//Kommunikáció nyitás
IF NOT(GVL.bLaserCommOpen) THEN
	LaserSocketOpen(
		sSrvNetId:= '', 
		sRemoteHost:= sLaserRemoteHost, 
		nRemotePort:= 20001, 
		bExecute:= bLaserSocketOpenEnable, 
		tTimeout:= T#45S, 
		bBusy=> bLaserSocketbusy, 
		bError=> bLaserSocketError, 
		nErrId=> nLaserSocketErrId, 
		hSocket=> hLaserSocket);
	IF bLaserSocketOpenEnable THEN
		IF (NOT(bLaserSocketError) AND NOT(bLaserSocketError) AND NOT(bLaserSocketbusy)) THEN
			bLaserSocketOpenEnable := FALSE;
			GVL.bLaserCommOpen:=TRUE;
			LaserSocketOpen(
				sSrvNetId:= '', 
				sRemoteHost:= sLaserRemoteHost, 
				nRemotePort:= 5000, 
				bExecute:= FALSE, 
				tTimeout:= T#45S, 
				bBusy=> bLaserSocketbusy, 
				bError=> bLaserSocketError, 
				nErrId=> nLaserSocketErrId, 
				hSocket=> hLaserSocket);
		ELSE
			IF NOT(bLaserSocketbusy) THEN
				bLaserSocketOpenEnable:=FALSE;
			END_IF
		END_IF
	ELSE
		bLaserSocketOpenEnable:=TRUE;
	END_IF
END_IF

// Parancsfordítások a lézer számára
IF bLaserSendReady=TRUE THEN				// a parancsküldés befejeződött,
	IF s_InCommand='GETJOB' THEN
		sLaserSend:='GetJob;';
	END_IF
	IF s_InCommand='START' THEN
		sLaserSend:='Start;';
	END_IF
	IF s_InCommand='SETTYPE' THEN
		s_TypeCode:=TO_STRING(GVL.iSelectedProductType);
		sLaserSend:=CONCAT('SetVars;TypeCode;',CONCAT(s_TypeCode,';'));
	END_IF
	IF s_InCommand='GETSTATUS' THEN
		sLaserSend:='GetStatus;';
	END_IF
	IF s_InCommand='RECEIVE' THEN
		bLaserSocketReceiveRequest:=TRUE;
		bLaserSendReady:=FALSE;
		sLaserReceived:='';
	END_IF
END_IF

// Csak akkor próbáljon kommunikálni, ha már megnyílt a kapcsolat
IF GVL.bLaserCommOpen=TRUE THEN
	// Adatküldés, ha van mit küldeni
	IF sLaserSend<>'' THEN
		IF bLaserSocketSendEnable THEN
			bLaserSocketSendEnable:=FALSE;
			sLaserSend:='';
			bLaserSocketReceiveRequest:=TRUE; // Választ is várunk majd a lézertől.
		ELSE
			MEMSET(ADR(baReceivedByteArray), 0, 256);
			MEMSET(ADR(baSendByteArray), 0, 256);
			baSendByteArray := MAXSTRING_TO_BYTEARR(sLaserSend);
			uSendByteLen := INT_TO_UDINT(LEN(sLaserSend));
			baSendByteArray[uSendByteLen]:=16#D;
			baSendByteArray[uSendByteLen+1]:=16#A;
			bLaserSocketSendEnable:=TRUE;
			bLaserSendReady:=FALSE;
			sLaserReceived:='';
		END_IF;
		LaserSocketSend(
			sSrvNetId:= '', 
			hSocket:= hLaserSocket, 
			cbLen:= uSendByteLen + 2, 
			pSrc:= ADR(baSendByteArray), 
			bExecute:= bLaserSocketSendEnable, 
			tTimeout:= T#5S, 
			bBusy=> bLaserSocketbusy, 
			bError=> bLaserSocketError, 
			nErrId=> nLaserSocketErrId);
	END_IF
	// Ha van adatfogadási igény, akkor minden páros ciklusnál indítson adatfogadást
	IF (bLaserSocketReceiveRequest=TRUE) AND (bEvenCycle=TRUE) THEN
		bLaserSocketReceiveEnable:=TRUE;
	ELSE
		bLaserSocketReceiveEnable:=FALSE;		
	END_IF
	//Adatfogadás, ha van rá parancs
	LaserSocketReceive(
		sSrvNetId:= '', 
		hSocket:= hLaserSocket, 
		cbLen:= 255, 
		pDest:= ADR(baReceivedByteArray), 
		bExecute:= bLaserSocketReceiveEnable, 
		tTimeout:= T#5S, 
		bBusy=> bLaserSocketbusy, 
		bError=> bLaserSocketError, 
		nErrId=> nLaserSocketErrId, 
		nRecBytes=> nLaserReceivedBytesNum);
	IF baReceivedByteArray[0]>0 THEN // Ha érkezett válasz a lézertől, akkor
		nLaserReceivedBytesNum:=0;	// töröljük, hogy ne lépjen be ide újra,
		bLaserSocketReceiveRequest:=FALSE;	// ne várjon több válaszra,		
		bLaserSendReady:=TRUE;				// a parancsküldés befejeződött, töröljük a parancsot, és
		bLaserSendOK:=(baReceivedByteArray[0]=16#6); // ha ACK jel jött, akkor OK.
		sLaserReceived := BYTEARR_TO_MAXSTRING(baReceivedByteArray);
		IF sLaserReceived='$06;0000;$R$N' THEN
			s_InCommand:='';
		ELSE
			s_InCommand:=CONCAT('LÉZER HIBA: ',sLaserReceived);
		END_IF
	END_IF

	//Kommunikáció bontás
	LaserSocketClose(
		sSrvNetId:= '', 
		hSocket:= hLaserSocket, 
		bExecute:= bLaserSocketCloseEnable, 
		tTimeout:= T#45S, 
		bBusy=> bLaserSocketbusy, 
		bError=> bLaserSocketError, 
		nErrId=> nLaserSocketErrId);

	bEvenCycle:=NOT bEvenCycle;
END_IF

END_PROGRAM

// ---- POUs/PISTI/Components/TEST_R_INTERPOL.TcPOU
PROGRAM TEST_R_INTERPOL
VAR
	rRNTC_MIN0, rRNTC_MIN1, rRNTC_MAX0, rRNTC_MAX1, rPt_MIN, rPt_MAX, rT: REAL;
END_VAR

rRNTC_MIN0:=f_GetNTCMinR(rTemp:=rT, nProd:=0);
rRNTC_MAX0:=f_GetNTCMaxR(rTemp:=rT, nProd:=0);
rRNTC_MIN1:=f_GetNTCMinR(rTemp:=rT, nProd:=1);
rRNTC_MAX1:=f_GetNTCMaxR(rTemp:=rT, nProd:=1);
rPt_MIN:=f_GetPtMinR(rTemp:=rT);
rPt_MAX:=f_GetPtMaxR(rTemp:=rT);

END_PROGRAM

// ---- POUs/PISTI/Helpers/f_GetNTCNomR.TcPOU
FUNCTION f_GetNTCNomR : real
VAR_INPUT
	rTemp: REAL;
	nProd: UINT;
END_VAR
VAR
	nI: INT;
	rT0, rT1, rR0, rR1, rM: REAL;
END_VAR
VAR CONSTANT
	rCorr: REAL := 1.1;
	NTC_Sensing_MinRT: ARRAY[0..1, 0..25] OF REAL := 
	[15, 16, 17, 18, 19, 20, 21, 22, 23, 24, 25, 26, 27, 28, 29, 30, 31, 32, 33, 34, 35, 36, 37, 38, 39, 40,
	14966.9, 14299.6, 13665.8, 13063.7, 12491.4, 11947.3, 11430, 10937.9, 10469.8, 10024.2, 9600, 9188.1, 8796.1, 8423, 8067.6, 7729.2, 7406.8, 7099.6, 6806.7, 6527.5, 6261.3, 6007.2, 5764.9, 5533.6, 5312.7, 5101.9];
	NTC_GE_MinRT: ARRAY[0..1, 0..23] OF REAL := 
	[15, 16, 17, 18, 19, 20, 21, 22, 23, 24, 25, 26, 27, 28, 29, 30, 31, 32, 33, 34, 35, 36, 38, 40,
	15133, 14457, 13815, 13206, 12626, 12075, 11552, 11053, 10579, 10128, 9700, 9279.9, 8883.4, 8506.1, 8146.8, 7804.7, 7478.7, 7168.1, 6872.1, 6589.9, 6320.7, 6064, 5585.4, 5149.3];
END_VAR

nI:=1;
(*IF nProd=0 THEN
	WHILE (NTC_Sensing_MinRT[0,nI]<rTemp) AND (nI<25) DO
		nI:=nI+1;
	END_WHILE
	rT0:=NTC_Sensing_MinRT[0,nI-1];
	rT1:=NTC_Sensing_MinRT[0,nI];
	rR0:=NTC_Sensing_MinRT[1,nI-1];
	rR1:=NTC_Sensing_MinRT[1,nI];
	rM:=(rR1-rR0)/(rT1-rT0);
	f_GetNTCMinR:=rR0+rM*(rTemp-rT0);
ELSE
	WHILE (NTC_GE_MinRT[0,nI]<rTemp) AND (nI<23) DO
		nI:=nI+1;
	END_WHILE
	rT0:=NTC_GE_MinRT[0,nI-1];
	rT1:=NTC_GE_MinRT[0,nI];
	rR0:=NTC_GE_MinRT[1,nI-1];
	rR1:=NTC_GE_MinRT[1,nI];
	rM:=(rR1-rR0)/(rT1-rT0);
	f_GetNTCMinR:=rR0+rM*(rTemp-rT0);	
END_IF*)
WHILE (GVL.NTC_Sensing_NomRT[0,nI]<rTemp) AND (nI<25) DO
	nI:=nI+1;
END_WHILE
rT0:=GVL.NTC_Sensing_NomRT[0,nI-1];
rT1:=GVL.NTC_Sensing_NomRT[0,nI];
rR0:=GVL.NTC_Sensing_NomRT[1,nI-1];
rR1:=GVL.NTC_Sensing_NomRT[1,nI];
rM:=(rR1-rR0)/(rT1-rT0);
f_GetNTCMinR:=(rR0+rM*(rTemp-rT0))/(1+GVL.rNTCDev/100);

END_FUNCTION

// ---- POUs/PISTI/Helpers/f_GetPtNomR.TcPOU
FUNCTION f_GetPtNomR : real
VAR_INPUT
	rTemp: REAL := 25;
END_VAR
VAR
	nI: INT;
	rT0, rT1, rR0, rR1, rM: REAL;
END_VAR
VAR CONSTANT
	Pt_MinRT: ARRAY[0..1, 0..15] OF REAL := 
	[0,20,40,60,80,100,120,140,160,180,200,220,240,260,280,300,
	990,1067,1143,1219,1294,1368,1442,1516,1588,1661,1733,1804,1875,1945,2015,2084];
END_VAR

nI:=1;
WHILE (Pt_MinRT[0,nI]<rTemp) AND (nI<15) DO
	nI:=nI+1;
END_WHILE
rT0:=Pt_MinRT[0,nI-1];
rT1:=Pt_MinRT[0,nI];
rR0:=Pt_MinRT[1,nI-1];
rR1:=Pt_MinRT[1,nI];
rM:=(rR1-rR0)/(rT1-rT0);
f_GetPtMinR:=rR0+rM*(rTemp-rT0);

END_FUNCTION

// ---- POUs/PISTI/Helpers/f_GetPtTfromR.TcPOU
FUNCTION f_GetPtTfromR : real
VAR_INPUT
	rR: REAL;
END_VAR
VAR
	nI: INT;
	rT0, rT1, rR0, rR1, rM: REAL;
END_VAR
VAR CONSTANT
	Pt_RT: ARRAY[0..1, 0..15] OF REAL := 
	[0,20,40,60,80,100,120,140,160,180,200,220,240,260,280,300,
	1000,1077.9,1155.4,1232.4,1309,1385.1,1460.7,1535.8,1610.5,1684.8,1758.6,1831.9,1904.7,1977.1,2049.1,2120.5];
END_VAR

nI:=1;
WHILE (Pt_RT[1,nI]<rR) AND (nI<15) DO
	nI:=nI+1;
END_WHILE
rT0:=Pt_RT[0,nI-1];
rT1:=Pt_RT[0,nI];
rR0:=Pt_RT[1,nI-1];
rR1:=Pt_RT[1,nI];
rM:=(rT1-rT0)/(rR1-rR0);
f_GetPtTfromR:=rT0+rM*(rR-rR0);

END_FUNCTION

// ---- POUs/PISTI/Helpers/f_GetISOLvalue.TcPOU
FUNCTION f_GetISOLvalue : REAL
VAR_INPUT
	rVoltage : REAL;
END_VAR
VAR
	rVoltagePerOhmRate : REAL := 5100/0.889;
END_VAR

f_GetISOLvalue := rVoltage * rVoltagePerOhmRate;

END_FUNCTION

// ---- GlobalTextList.TcGTLO
TEXTLIST GlobalTextList
  140 = ''
  845 = '\nFizikális gombok használata NTC vágáshoz.\nZöld gomb: NTC vágófej le-fel\nPiros gomb: NTC vágófej le-fel'
  844 = '\nFizikális gombok használata NTC vágáshoz.Zöld gomb: NTC vágófej le-fel\nPiros gomb: NTC vágófej le-fel'
  841 = '\nZöld gomb: NTC vágófej le-fel\nPiros gomb: NTC vágófej le-fel'
  842 = '\nZöld gomb: NTC vágás\nPiros gomb: NTC elengedés'
  840 = '\nZöld gomb: NTC vágófej le-fel\nPiros gomb: NTC vágófej le-fel'
  43 = '%'
  47 = '%./100'
  45 = '%.1f'
  46 = '%.2f'
  48 = '%/100'
  157 = '%c'
  130 = '%d'
  60 = '%f'
  59 = '%lr'
  58 = '%s'
  73 = '%u'
  368 = "'ELEKTRÓDA$R$NCSERE!'"
  49 = '.1f'
  2499 = '1. elektróda pár'
  807 = '1. elektródapár'
  717 = '1. heg.'
  380 = '1. HEGESZTESHEZ'
  390 = '1. hegesztés program'
  384 = '1. HEGESZTÉSHEZ'
  800 = '1. VÉGPOZÍCIÓ'
  802 = '1. VÉGPOZÍCIÓHOZ'
  41 = '11'
  44 = '1f'
  7390 = '2. elektróda pár'
  809 = '2. elektródapár'
  718 = '2. heg.'
  381 = '2. HEGESZTESHEZ'
  391 = '2. hegesztés program'
  385 = '2. HEGESZTÉSHEZ'
  801 = '2. VÉGPOZÍCIÓHOZ'
  5960 = '3. elektróda pár'
  808 = '3. elektródapár'
  719 = '3. heg.'
  382 = '3. HEGESZTESHEZ'
  392 = '3. hegesztés program'
  386 = '3. HEGESZTÉSHEZ'
  317 = '4. heg.'
  287 = '4. heg. deformációja:'
  383 = '4. HEGESZTESHEZ'
  708 = '4. hegesztés'
  286 = '4. hegesztés deformációja:'
  393 = '4. hegesztés program'
  710 = '4. hegesztés, STOP érték [um]:'
  387 = '4. HEGESZTÉSHEZ'
  318 = '5. heg.'
  288 = '5. heg. deformációja:'
  709 = '5. hegesztés'
  394 = '5. hegesztés program'
  711 = '5. hegesztés, STOP érték [um]:'
  388 = '5. HEGESZTÉSHEZ'
  484 = '6 s'
  729 = '6. hegesztés program'
  341 = '6.0'
  116 = '600V'
  115 = '600VBe'
  117 = '600VExt'
  314 = '637 GYÁRTÓ CELLA'
  6089 = '637900'
  730 = '7. hegesztés program'
  9321 = '745900'
  7231 = '745910'
  830 = '<!> db'
  509 = 'A jelölö lézer saját vezérlö szoftvere'
  504 = 'A jelölő lézer saját vezérlő szoftvere'
  901 = 'A Pt oldali kamera saját vezérlő szoftvere'
  637 = 'A tengelypozíciók a megfelelö\nszervízfüleken állíthatók be.\n\nAz alábbi gombok a megfelelö \nszervízfülre navigálnak:'
  625 = 'A tengelypozíciók a megfelelő\nszervízfüleken állíthatók be.\n\nAz alábbi gombok a megfelelő \nszervízfülre navigálnak:'
  619 = 'A tengelypozíciók a megfelelő\nszervízfüleken állíthatók be.\nAz alábbi gombok a\nmegfelelő szervízfülre\nnavigálnak:'
  620 = 'A tengelypozíciók a megfelelő\nszervízfüleken állíthatók be.\nAz alábbi gombok a \nmegfelelő szervízfülre\nnavigálnak:'
  622 = 'A tengelypozíciók a megfelelő\nszervízfüleken állíthatók be.\nAz alábbi gombok a megfelelő\nszervízfülre\nnavigálnak:'
  623 = 'A tengelypozíciók a megfelelő\nszervízfüleken állíthatók be.\nAz alábbi gombok a megfelelő \nszervízfülre\nnavigálnak:'
  624 = 'A tengelypozíciók a megfelelő\nszervízfüleken állíthatók be.\nAz alábbi gombok a megfelelő \nszervízfülre navigálnak:'
  621 = 'A tengelypozíciók a megfelelő\nszervízfüleken állíthatók be.\nAz alábbi gombok a megfelelő szervízfülre\nnavigálnak:'
  618 = 'A tengelypozíciók a megfelelő szervízfüleken állíthatók be. Az alábbi gombok a megfelelő szervízfülre navigálnak:'
  62 = 'Act. Pos:'
  8 = 'AdapterLefogó'
  544 = 'Adapterlefogó'
  5 = 'AdapterLefogóBent'
  4 = 'AdapterLefogóKint'
  818 = 'Adapterérzékelö'
  2 = 'Adapterérzékelő'
  917 = 'ADD/DELETE USER'
  300 = 'Admin'
  79 = 'AEH'
  1962 = 'AJTÓ\nZÁR'
  692 = 'Ajtók zárva'
  143 = 'ALARM'
  352 = 'Alsó rész'
  179 = 'AUTO'
  285 = 'AUTO STOP'
  488 = 'Automata'
  713 = 'Automatikus mentés'
  81 = 'AVH'
  771 = 'bal fent'
  832 = 'Bal fék'
  772 = 'bal lent'
  838 = 'Bal lábérzékelö'
  833 = 'Bal lábérzékelő'
  425 = 'Bal pofa'
  105 = 'Balon'
  436 = 'Balra'
  439 = 'Be'
  20 = 'Behelyezés'
  547 = 'BEHELYEZÉS'
  668 = 'Belépve, mint:'
  669 = 'BELÉPVE, MINT:'
  107 = 'Bent'
  591 = 'Beragadt TCP IP kapcsolatok törölve'
  97 = 'Bereit'
  465 = 'BEZÁR'
  826 = 'BEÁLLÍTÁS'
  348 = 'Beállítások'
  714 = 'Beállítások automatikus mentése'
  682 = 'BIZTONSÁGI AJTÓ RETESZ'
  679 = 'Biztonsági kör OK'
  678 = 'Biztonsági relé föld OK'
  677 = 'Biztonsági relé táp OK'
  676 = 'Biztonsági rendszer'
  4978 = 'Biztos?'
  876 = 'Busy'
  900 = 'Checker indítása'
  794 = 'Ciklusok'
  160 = 'CLOSE'
  122 = 'Com Open'
  878 = 'Comm Open'
  266 = 'COMMUNICATION OPEN'
  865 = 'Csatlakozó'
  4888 = 'Csatlakozó\nfedél csukva'
  491 = 'Csatlakozó\nfedél nyitva'
  6459 = 'Csatlakozó\nfedél zárva'
  866 = 'Csatlakozó (745)'
  864 = 'Csatlakozó fedél'
  490 = 'Csatlakozó fedél edelNyitva?'
  532 = 'CSIPESZ NYIT'
  531 = 'CSIPESZ ZÁR'
  277 = 'DARABSZÁM'
  812 = 'db'
  707 = 'Deformációalapú hegesztés-leállítás'
  4104 = 'Dolgozói szám'
  814 = 'Elekróda karbantartás'
  805 = 'ELEKT-\nRÓDA-\nTISZTÍTÁS'
  208 = 'Elektroden\nAnfordem'
  96 = 'ElektrodenAnfordem'
  364 = 'ELEKTRÓDA  CSERE!'
  363 = 'ELEKTRÓDA CSERE!'
  365 = 'ELEKTRÓDA RÉGI'
  366 = 'ELEKTRÓDA$R$NCSERE!'
  370 = 'ELEKTRÓDACSERE'
  369 = 'ELEKTRÓDACSERE!'
  803 = 'ELEKTRÓDATISZT'
  804 = 'ELEKTRÓDATISZTÍTÁS'
  367 = 'ELEKTRÓDA\\R\\NCSERE!'
  907 = 'ELFOGADHATÓ'
  222 = 'ELLENALLAS'
  252 = 'ELLENALLAS ETALON'
  450 = 'ELLENÁLLÁS'
  452 = 'Ellenállás'
  451 = 'ELLENÁLLÁS ETALON'
  658 = 'Eltelt idö'
  480 = 'Eltelt idö (s)'
  513 = 'Elvárt kód:'
  469 = 'ELVÁRT:'
  379 = 'Elvégzendö müveletek'
  347 = 'Elvégzendö műveletek'
  516 = 'ELÖHAJLÍTASHOZ'
  424 = 'ELÖHAJLÍTÁS'
  517 = 'ELÖHAJLÍTÁSHOZ'
  349 = 'Elöhajlító'
  83 = 'ELŐHAJLITASHOZ'
  194 = 'ELŐHAJLÍTÁS'
  76 = 'Előhajlító'
  77 = 'Előhajlító fent'
  546 = 'Enged'
  701 = 'EPSON RC+ megnyitása'
  410 = 'Eredmény:'
  466 = 'EREDMÉNYEK'
  174 = 'ERROR'
  246 = 'Error'
  877 = 'Error ID'
  283 = 'Error reset'
  175 = 'ESTOP'
  695 = 'Etalon'
  556 = 'Etalon mérés'
  694 = 'ETALON MÉRÉS'
  109 = 'FedelLecsukva?'
  249 = 'FedelNyitva?'
  829 = 'FEDÉL'
  78 = 'FEH'
  431 = 'Fej le'
  670 = 'FEJLESZTÖ'
  716 = 'Felfüggeszt'
  350 = 'Felsö rész'
  103 = 'Fent'
  779 = 'fent'
  775 = 'fent bent'
  776 = 'fent kint'
  725 = 'Fizikális gombok használata NTC vágáshoz.\nZöld gomb: NTC vágás\nPiros gomb: NTC elengedés'
  846 = 'Fizikális gombok használata NTC vágáshoz.\nZöld gomb: NTC vágófej le-fel\nPiros gomb: NTC vágófej le-fel'
  503 = 'FOBA Draw indítása'
  268 = 'Fogadott:'
  269 = 'Fogadás'
  42 = 'fok'
  690 = 'FOLYTAT'
  554 = 'Forgásirány:'
  149 = 'Forward'
  909 = 'FRISSÍT'
  80 = 'FVH'
  3 = 'Fénykapu'
  674 = 'FÉNYSOROMPÓ'
  434 = 'Fütötömb'
  527 = 'Fütötömb\nfelfütött'
  478 = 'Fütötömb beállított\nhömérséklete (C)'
  615 = 'Fütötömb beállított\nhömérséklete (C):'
  656 = 'Fütötömb beállított\nhömérséklete [C]'
  644 = 'Fütötömb beállított \nhömérséklete (C):'
  650 = 'Fütötömb beállított \nhömérséklete [C]:'
  477 = 'Fütötömb hömérséklete (C)'
  67 = 'Főnök'
  530 = 'GroupBox'
  291 = 'Hajlítás'
  354 = 'Hajlítók'
  316 = 'Heg. deformációja:'
  904 = 'Hegesz-\ntéshez'
  795 = 'HEGESZ-\nTÖFEJ\nTISZTÍTÁS'
  903 = 'Hegesz-téshez'
  85 = 'HEGESZTES1HEZ'
  87 = 'HEGESZTES2HOZ'
  86 = 'HEGESZTES2HÖZ'
  88 = 'HEGESZTES3HOZ'
  89 = 'HEGESZTES4HEZ'
  90 = 'HEGESZTES5HÖZ'
  138 = 'HEGESZTESHEZ'
  216 = 'HEGESZTESHEZ1'
  217 = 'HEGESZTESHEZ2'
  21 = 'Hegesztés'
  74 = 'HEGESZTÉS'
  791 = 'HEGESZTÉS KÉSZ'
  292 = 'Hegesztés1'
  627 = 'HEGESZTÉS1'
  519 = 'HEGESZTÉS1-HEZ'
  293 = 'Hegesztés2'
  628 = 'HEGESZTÉS2'
  520 = 'HEGESZTÉS2-HÖZ'
  294 = 'Hegesztés3'
  629 = 'HEGESZTÉS3'
  521 = 'HEGESZTÉS3-HOZ'
  295 = 'Hegesztés4'
  630 = 'HEGESZTÉS4'
  522 = 'HEGESZTÉS4-HEZ'
  296 = 'Hegesztés5'
  631 = 'HEGESZTÉS5'
  523 = 'HEGESZTÉS5-HÖZ'
  305 = 'Hegesztés6'
  306 = 'Hegesztés7'
  902 = 'Hegesztéshez'
  588 = 'Hegesztö'
  799 = 'Hegesztö elektróda karbantartás'
  407 = 'Hegesztö státusz'
  579 = 'Hegesztö üzemkész'
  459 = 'HEGESZTÖFEJ\nTISZTÍTÁS'
  781 = 'Hegesztöfej I/O-k'
  400 = 'HEGESZTÖFEJ TISZT.'
  783 = 'Hegesztöfej1'
  757 = 'Hegesztöfej1 bal fent'
  761 = 'Hegesztöfej1 bal lent'
  758 = 'Hegesztöfej1 jobb fent'
  762 = 'Hegesztöfej1 jobb lent'
  755 = 'Hegesztöfej1 le'
  765 = 'Hegesztöfej1 útmérö:'
  784 = 'Hegesztöfej2'
  756 = 'Hegesztöfej2 be'
  763 = 'Hegesztöfej2 fent bent'
  759 = 'Hegesztöfej2 fent kint'
  770 = 'Hegesztöfej2 ki'
  764 = 'Hegesztöfej2 lent bent'
  760 = 'Hegesztöfej2 lent kint'
  766 = 'Hegesztöfej2 útmérö:'
  785 = 'Hegesztöfej3'
  768 = 'Hegesztöfej3 fent'
  767 = 'Hegesztöfej3 le'
  769 = 'Hegesztöfej3 lent'
  593 = 'Hegesztöfejek alapállapotban'
  356 = 'Hegesztögép státusza'
  9 = 'Hegesztő'
  68 = 'Hegesztő1'
  71 = 'Hegesztő1 Útmérő:'
  735 = 'Hegesztő1 útmérő:'
  69 = 'Hegesztő2'
  72 = 'Hegesztő2 Útmérő:'
  736 = 'Hegesztő2 útmérő:'
  70 = 'Hegesztő3'
  274 = 'HEGESZTŐFEJ TISZT.'
  739 = 'Hegesztőfej1 bal fent'
  740 = 'Hegesztőfej1 bal lent'
  743 = 'Hegesztőfej1 fent kint'
  741 = 'Hegesztőfej1 jobb fent'
  742 = 'Hegesztőfej1 jobb lent'
  750 = 'Hegesztőfej1 le'
  737 = 'Hegesztőfej1 útmérő:'
  751 = 'Hegesztőfej2 be'
  745 = 'Hegesztőfej2 fent bent'
  744 = 'Hegesztőfej2 fent kint'
  747 = 'Hegesztőfej2 lent bent'
  746 = 'Hegesztőfej2 lent kint'
  738 = 'Hegesztőfej2 útmérő:'
  753 = 'Hegesztőfej3 bal fent'
  754 = 'Hegesztőfej3 bal lent'
  748 = 'Hegesztőfej3 fent'
  752 = 'Hegesztőfej3 le'
  749 = 'Hegesztőfej3 lent'
  6 = 'HegesztőFent'
  7 = 'HegesztőLent'
  782 = 'Hello'
  732 = 'HIBA'
  398 = 'Hiba kód:'
  399 = 'Hiba törlés'
  403 = 'Hiba törlése'
  401 = 'Hibakód:'
  404 = 'Hibatörlés'
  733 = 'HIBATÖRLÉS'
  279 = 'HIBÁS'
  857 = 'Himba'
  867 = 'Himba alapállapotban'
  858 = 'Himba be'
  860 = 'Himba elöl'
  861 = 'Himba hátul'
  870 = 'Himba OK'
  863 = 'Himba pozíció'
  859 = 'Himba érzékelő'
  862 = 'HIMBÁHOZ'
  53 = 'HOME'
  449 = 'HÖM (C)'
  332 = 'HÖM [C]'
  529 = 'Hömérséklet (C)'
  910 = 'Hüvely poz OK'
  911 = 'Hüvely pozíció'
  912 = 'Hüvely van'
  721 = 'Hüvelyek OK'
  448 = 'HŐM (C)'
  321 = 'HŐM MEAS (C)'
  214 = 'Hőmérséklet'
  218 = 'Hőmérséklet (C)'
  224 = 'IDOALLANDO'
  250 = 'IDOALLANDO_OK'
  323 = 'IDÖÁLLANDÓ'
  485 = 'Idöállandó'
  642 = 'Idöállandó\nfelsö határa:'
  616 = 'Idöállandó\nfelső határa:'
  647 = 'Idöállandó \nfelsö határa (s):'
  648 = 'Idöállandó \nfelsö határa [s]:'
  645 = 'Idöállandó \nfelsö határa:'
  481 = 'Idöállandó (s)'
  328 = 'IDÖÁLLANDÓ [s]'
  654 = 'Idöállandó [s]'
  298 = 'IDÖÁLLANDÓ_OK'
  242 = 'Időállandó (s)'
  4983 = 'IGEN'
  789 = 'In-Sight Explorer indítása'
  358 = 'INDÍTÁS'
  817 = 'Indítás fénysorompóval'
  787 = 'Indítási feltételek'
  585 = 'Indítási opciók'
  170 = 'INIT'
  324 = 'ISOL'
  221 = 'ISOL_OK'
  672 = 'IV-Navigator indítása'
  223 = 'IZOLÁCIÓ'
  114 = 'Izolációs érték'
  243 = 'Izolációs érték (V)'
  232 = 'Izolációs érték(V)'
  311 = 'JELENLEGI FOLYAMAT:'
  389 = 'Jelenlegi pozíció:'
  825 = 'Jelenlegi érték [%]:'
  824 = 'Jelenlegi érték [0...100 %]:'
  325 = 'JELÖLÉS'
  297 = 'JELÖLÉS_OK'
  773 = 'jobb fent'
  835 = 'Jobb fék'
  774 = 'jobb lent'
  839 = 'Jobb lábérzékelö'
  834 = 'Jobb lábérzékelő'
  426 = 'Jobb pofa'
  106 = 'Jobbon'
  55 = 'JOG +'
  56 = 'JOG -'
  4109 = 'Jogosultság'
  181 = 'JozsiProcess.asActualProgram[0,INDEX]'
  182 = 'JozsiProcess.asActualProgram[1,INDEX]'
  183 = 'JozsiProcess.asActualProgram[2,INDEX]'
  184 = 'JozsiProcess.asActualProgram[3,INDEX]'
  185 = 'JozsiProcess.asActualProgram[4,INDEX]'
  186 = 'JozsiProcess.asActualProgram[5,INDEX]'
  64 = 'JozsiTengely'
  278 = 'JÓ'
  24 = 'Józsi'
  604 = 'Kamera'
  728 = 'KAMERA'
  895 = 'Kamera Adapter'
  893 = 'Kamera All pass'
  894 = 'Kamera Any fail'
  886 = 'Kamera Aquiring'
  890 = 'Kamera Inspect toggle'
  889 = 'Kamera Inspecting'
  896 = 'Kamera Kappe'
  888 = 'Kamera Online'
  892 = 'Kamera Part Detected'
  727 = 'Kamera pozíció'
  897 = 'Kamera Pt'
  891 = 'Kamera Results available'
  898 = 'Kamera Run'
  882 = 'Kamera Set Offline'
  887 = 'Kamera Setup'
  881 = 'Kamera Trigger'
  885 = 'Kamera Trigger Ack'
  880 = 'Kamera Trigger EN'
  884 = 'Kamera Trigger Ready'
  723 = 'KAMERA-\nEREDMÉNYEK'
  610 = 'Kamera1'
  611 = 'Kamera2'
  722 = 'KAMERAEREDMÉNYEK'
  724 = 'Kameravizsgálat\neredménye'
  726 = 'KAMERÁHOZ'
  165 = 'KAPPE'
  251 = 'Kappe Pistikének'
  432 = 'Kappe prés'
  464 = 'KAPPE PRÉS'
  307 = 'Kappe, robot'
  15 = 'KappeBal'
  13 = 'KappeBalFent'
  14 = 'KappeBalLent'
  12 = 'KappeFelLe'
  10 = 'KappeFent'
  18 = 'KappeJobb'
  16 = 'KappeJobbFent'
  17 = 'KappeJobbLent'
  11 = 'KappeLent'
  337 = 'KappeNincsLent'
  137 = 'KAPPEZASHOZ'
  905 = 'Kappé-\nzáshoz'
  22 = 'Kappézás'
  634 = 'KAPPÉZÁS'
  525 = 'KAPPÉZÁSHOZ'
  798 = 'KARBANTARTÁS'
  855 = 'Keyence SR-1000W'
  856 = 'Keyence SR-1000W/ nem Zebra'
  693 = 'Ki'
  417 = 'Kieg. müveletek'
  416 = 'Kiegészítö müveletek'
  346 = 'KILÉPÉS'
  3792 = 'Kilépés'
  108 = 'Kint'
  152 = 'Kiszedo'
  376 = 'Kiszedö'
  351 = 'Kitol'
  299 = 'KIÉRTÉKELÉS'
  422 = 'Kommunikáció'
  557 = 'KOMMUNIKÁCIÓS CSATORNA MEGNYITVA'
  505 = 'KOMMUNIKÁCIÓS VONAL MEGNYITVA'
  608 = 'Kábeltáv OK'
  688 = 'Kérem, adja meg a vonalkód\nolvasó\nsegítségével a gyártani kívánt terméktípust!\nÜgyeljen rá, hogy a megfelelő NTC és Pt1000\nalkatrészek legyenek betárazva, felhasználva!\nHa kell, ezek vonalkódját is be lehet olvastatni.'
  687 = 'Kérem, adja meg a vonalkód\nolvasó segítségével\na \ngyártani kívánt terméktípust!\nÜgyeljen rá, hogy a megfelelő NTC és Pt1000\nalkatrészek legyenek betárazva, felhasználva!\nHa kell, ezek vonalkódját is be lehet olvastatni.'
  686 = 'Kérem, adja meg a vonalkód\nolvasó segítségével a \ngyártani kívánt terméktípust!\nÜgyeljen rá, hogy a megfelelő NTC és Pt1000 alkatrészek legyenek betárazva, felhasználva!\nEzek vonalkódját is be lehet olvastatni.'
  685 = 'Kérem, adja meg a vonalkód\nolvasó segítségével a \ngyártani kívánt terméktípust!\nÜgyeljen rá, hogy a megfelelő NTC és Pt1000 alkatrészek legyenek betárazva, felhasználva! Ezek vonalkódját is be lehet olvastatni.'
  684 = 'Kérem, adja meg a vonalkód\nolvasó segítségével a\ngyártani kívánt terméktípust!'
  689 = 'Kérem, adja meg a vonalkódolvasó\nsegítségével a gyártani kívánt terméktípust!\nÜgyeljen rá, hogy a megfelelő NTC és Pt1000\nalkatrészek legyenek betárazva, felhasználva!\nHa kell, ezek vonalkódját is be lehet olvastatni.'
  471 = 'Kérem, indítás elött ellenörízze,\nhogy idegen tárgyaktól\nmentes-e a munkatér, és\nminden készen áll-e az indításra!'
  470 = 'Kérem, indítás előtt ellenörízze,\nhogy idegen tárgyaktól\nmentes-e a munkatér, és\nminden készen áll-e az indításra!'
  699 = 'Kérem, tegye be a(z) %s. etalont,\nmajd nyomja meg a START gombot!'
  698 = 'Kérem, tegye be az %s. etalont,\nmajd nyomja meg a START gombot!'
  700 = 'Kérem, tegye be az ETALON%s-t,\nmajd nyomja meg a START gombot!'
  156 = 'Kérleltetés'
  372 = 'Késleltetés'
  359 = 'KÉSZ'
  395 = 'Készenléti program'
  444 = 'Kézi'
  823 = 'Kívánt érték [0...100 %]:'
  822 = 'Kívánt érték:'
  336 = 'Kódolvasó'
  514 = 'KÓDOLVASÓ'
  852 = 'KÓDOLVASÓ 2'
  333 = 'KÓDOLVASÓHOZ'
  853 = 'KÓDOLVASÓHOZ 2'
  256 = 'Következő lépés'
  272 = 'Közvetett parancs'
  273 = 'Közvetlen parancs'
  267 = 'Küld:'
  506 = 'kÜLDÉS'
  827 = 'KÜLDÉS'
  1 = 'Label'
  435 = 'Le'
  828 = 'LEKÉRDEZÉS'
  104 = 'Lent'
  780 = 'lent'
  777 = 'lent bent'
  778 = 'lent kint'
  335 = 'Leolvasott kód'
  512 = 'Leolvasott kód:'
  82 = 'LEVEGO'
  589 = 'Levegö'
  603 = 'LEVEGÖ'
  786 = 'Leállítási feltételek'
  120 = 'Load Recipe'
  125 = 'Login'
  141 = 'LOGIN'
  712 = 'Logolás'
  126 = 'Logout'
  564 = 'LOGOUT'
  7482 = 'Létezik'
  270 = 'Lézer'
  508 = 'LÉZER'
  592 = 'Lézer beállítva'
  673 = 'Lézer rendben'
  440 = 'Lézer takaró'
  578 = 'Lézer takaró zárva'
  821 = 'Lézer teljesítmény'
  309 = 'Lézerezés'
  507 = 'LÉZERHEZ'
  35 = 'LézerNyitva'
  37 = 'LézerNyitZár'
  595 = 'Lézerprogram beállítva'
  253 = 'LézerTakaró'
  36 = 'LézerZárva'
  284 = 'Mappa:'
  330 = 'MAX'
  811 = 'Max. db'
  613 = 'Max. szigetelési\nérték (V)'
  614 = 'Max. szigetelési\nérték (V):'
  643 = 'Max. szigetelési \nérték (V):'
  651 = 'Max. szigetelési \nérték [V]:'
  612 = 'Max. szigetelési érték (V)'
  653 = 'Max. szigetelési érték [V]'
  813 = 'max.db'
  657 = 'Megengedett max.\nidöállandó'
  639 = 'Megengedett max.\nidöállandó (s)'
  482 = 'Megengedett max. Idöállandó (s)'
  483 = 'Megengedett max. idöállandó (s)'
  153 = 'Megfogo'
  377 = 'Megfogó'
  691 = 'MEGSZAKÍT'
  92 = 'MELDUNG...'
  715 = 'Mentés'
  329 = 'MIN'
  94 = 'MITSTROM'
  99 = 'MitStrom'
  93 = 'MITSTROME'
  61 = 'MOVE'
  5238 = 'MOZOG'
  8518 = 'Mégse'
  331 = 'MÉRT'
  308 = 'Mérés'
  282 = 'Mérés reset'
  345 = 'Mérési eredmények'
  23 = 'MérésLézerezés'
  438 = 'Méröfej'
  704 = 'Mérötük Lent'
  34 = 'MérőBeKi'
  32 = 'MérőBent'
  437 = 'Mérőfej'
  40 = 'MérőfejBeKi'
  38 = 'MérőfejBent'
  39 = 'MérőfejKint'
  33 = 'MérőKint'
  454 = 'Müveletek tengely pozíciói:'
  453 = 'Müveletek Tengely pozíciók:'
  705 = 'Nagyfesz.\nMérötük Lent'
  706 = 'Nagyfesz.\nmérötük lent'
  4989 = 'NEM'
  908 = 'NEM JÓ'
  906 = 'NEM JÓ!'
  362 = 'NEM ÜZEMKÉSZ'
  100 = 'NichtBereit'
  8527 = 'Nincs ilyen felhasználó, olvassa be mégegyszer!'
  429 = 'Nincs lent'
  303 = 'None'
  193 = 'NTC'
  441 = 'NTC (Ohm)'
  446 = 'NTC (OHM)'
  234 = 'NTC CALC (C)'
  240 = 'NTC CALC (OHM)'
  703 = 'NTC elengedés'
  112 = 'NTC Ellenállás'
  219 = 'NTC Ellenállás (Ohm)'
  161 = 'NTC ELVEVÉS'
  412 = 'NTC ELVÉTEL'
  162 = 'NTC HEGESZTESHEZ'
  164 = 'NTC HEGESZTESTOL EL'
  4127 = 'NTC HEGESZTÉS'
  413 = 'NTC HEGESZTÉSHEZ'
  414 = 'NTC HEGESZTÉSTÖL EL'
  819 = 'NTC hütés'
  820 = 'NTC hütés\ntiltása'
  790 = 'NTC LÁBHAJLÍTÁS'
  233 = 'NTC MAX (C)'
  319 = 'NTC MAX (OHM)'
  241 = 'NTC MEAS (OHM)'
  211 = 'NTC Megfogo'
  263 = 'NTC Megfogó'
  235 = 'NTC MIDD (C)'
  236 = 'NTC MIN (C)'
  320 = 'NTC MIN (OHM)'
  405 = 'NTC oldal'
  680 = 'NTC oldali fénysorompó tilt'
  601 = 'NTC OLDALI TENGELY'
  831 = 'NTC pozícionálás'
  339 = 'NTC szerelés'
  397 = 'NTC szerelési oldal'
  231 = 'NTC TEMP CALC'
  229 = 'NTC TEMP MAX'
  230 = 'NTC TEMP MIN'
  586 = 'NTC tengely'
  569 = 'NTC tengely bekapcsolva'
  576 = 'NTC tengely bekapcsolásra kész'
  574 = 'NTC tengely HOME kész'
  572 = 'NTC tengely HOME rendben'
  567 = 'NTC tengely üzemkész'
  661 = 'NTC TÍPUS'
  662 = 'NTC TÍPUS:'
  563 = 'NTC türés [%]:'
  555 = 'NTC tűrés [%]:'
  702 = 'NTC vágás'
  374 = 'NTC vágó'
  2495 = 'NTC vágó Servo'
  326 = 'NTC [Ohm]'
  396 = 'NTC-s oldal'
  415 = 'NTC-VÁGÁS'
  463 = 'NTC-VÁGÓ'
  850 = 'NTC1 türés [%]:'
  849 = 'NTC2 (Ohm)'
  851 = 'NTC2 türés [%]:'
  854 = 'NTC2 [Ohm]'
  210 = 'NTCELENGEDÉS'
  209 = 'NTCVAGAS'
  213 = 'NTC_OK'
  338 = 'NULLÁZ'
  810 = 'NULLÁZÁS'
  443 = 'Nyit'
  154 = 'Nyitva'
  4100 = 'Név'
  447 = 'OK'
  916 = 'OLVAS'
  468 = 'OLVASOTT:'
  8509 = 'Olvassa be vonalkódját!'
  159 = 'OPEN'
  264 = 'OPEN COMM'
  302 = 'Operator'
  188 = 'Param1'
  189 = 'Param2'
  190 = 'Param3'
  191 = 'Param4'
  192 = 'Param5'
  132 = 'Paraméter1'
  133 = 'Paraméter2'
  134 = 'Paraméter3'
  135 = 'Paraméter4'
  136 = 'Paraméter5'
  187 = 'Parancs'
  510 = 'Parancs lista megnyitása'
  173 = 'PAUSED'
  163 = 'PIHI'
  479 = 'Pillanatnyi hömérséklet (C)'
  655 = 'Pillanatnyi hömérséklet [C]'
  837 = 'Piros gomb'
  25 = 'Pisti'
  65 = 'PistiTengely'
  30 = 'PlatniBalon'
  28 = 'PlatniFelLe'
  27 = 'PlatniFent'
  31 = 'PlatniForgat'
  29 = 'PlatniJobbon'
  433 = 'PlatniLe'
  26 = 'PlatniLent'
  373 = 'Pneumatikus mozgató egységek'
  430 = 'Pofák fel/le'
  495 = 'Pozíció:'
  128 = 'Program'
  198 = 'Program1HG1'
  199 = 'Program2HG1'
  200 = 'Program3HG1'
  205 = 'Program4HG1'
  201 = 'Program4HG2'
  202 = 'Program5HG2'
  206 = 'Program6HG2'
  203 = 'Program6HG3'
  204 = 'Program7HG3'
  207 = 'Program8HG3'
  428 = 'Prés fej'
  427 = 'Présel'
  788 = 'Pt hegesztés OK'
  872 = 'Pt Kamera'
  899 = 'Pt Kamera alapállapotban'
  515 = 'Pt oldal'
  734 = 'Pt oldali kamera'
  599 = 'Pt OLDALI TENGELY'
  322 = 'PT1000'
  442 = 'PT1000 (Ohm)'
  445 = 'PT1000 (OHM)'
  113 = 'PT1000 Ellenállás'
  220 = 'PT1000 Ellenállás (Ohm)'
  467 = 'Pt1000 hömérséklet változása'
  342 = 'Pt1000 hőmérséklet változása'
  227 = 'PT1000 MAX'
  237 = 'PT1000 MAX (OHM)'
  659 = 'PT1000 MAX [Ohm]'
  226 = 'PT1000 MEAS'
  238 = 'PT1000 MEAS (OHM)'
  225 = 'PT1000 MIN'
  239 = 'PT1000 MIN (OHM)'
  502 = 'PT1000 MÉRT (OHM)'
  660 = 'PT1000 MÉRT [Ohm]'
  228 = 'PT1000 NTC TEMP MAX'
  406 = 'Pt1000 oldal'
  681 = 'Pt1000 oldali fénysorompó tilt'
  731 = 'Pt1000 oldali kamera'
  600 = 'Pt1000 OLDALI TENGELY'
  340 = 'Pt1000 szerelés'
  402 = 'Pt1000 szerelési oldal'
  587 = 'Pt1000 tengely'
  570 = 'Pt1000 tengely bekapcsolva'
  577 = 'Pt1000 tengely bekapcsolásra kész'
  573 = 'Pt1000 tengely HOME kész'
  568 = 'Pt1000 tengely üzemkész'
  663 = 'Pt1000 TÍPUS:'
  638 = 'Pt1000 türés [%]:'
  327 = 'PT1000 [Ohm]'
  212 = 'PT1000_OK'
  129 = 'PTR'
  167 = 'RC'
  168 = 'RE'
  142 = 'Ready'
  171 = 'READY'
  166 = 'RELAX'
  584 = 'RENDSZER'
  683 = 'Rendszer'
  602 = 'Rendszer indulási állapota'
  304 = 'Rendszer indítása'
  583 = 'Rendszer állapota'
  598 = 'Rendszerindítás'
  581 = 'Rendszerindítás\nkihagyása'
  147 = 'Reset'
  582 = 'RESET'
  57 = 'RESET ERROR'
  150 = 'Reverse'
  111 = 'RL_ISOL'
  50 = 'Robot'
  462 = 'ROBOT'
  3364 = 'ROBOT HOME'
  537 = 'Robot kari eszközök'
  549 = 'Robot koordináták'
  575 = 'Robot kész'
  457 = 'Robot müveletek'
  411 = 'Robot műveletek'
  5345 = 'ROBOT OK'
  421 = 'Robot program:'
  566 = 'Robot rendben'
  7634 = 'ROBOT RUNNING'
  409 = 'Robot státusz'
  596 = 'Robot tengelyektöl távol'
  456 = 'Robot vezérlö:'
  420 = 'Robot vezérlő:'
  419 = 'Robot vezérlő:E'
  792 = 'ROBOT VÉSZLEÁLLÍTÁS\nAKTIVÁLVA!'
  139 = 'ROBOTMUVELETHEZ'
  635 = 'ROBOTMÜVELET'
  418 = 'ROBOTMÜVELETHEZ'
  127 = 'RUN'
  172 = 'RUNNING'
  847 = 'RÉGI\nPANEL'
  473 = 'RÉGI PANEL'
  545 = 'Rögzít'
  606 = 'Rögzítés OK'
  176 = 'SAFEGUARD'
  66 = 'Sardi'
  254 = 'SARDISAJAT1'
  255 = 'SARDISAJAT2'
  121 = 'Save Recipe'
  101 = 'Semelyik'
  265 = 'SEND'
  883 = 'Send Byte 2'
  177 = 'SERROR'
  301 = 'Service'
  54 = 'SERVO'
  144 = 'Servo'
  124 = 'Servo Off'
  123 = 'Servo On'
  247 = 'SOKK'
  476 = 'Sokk'
  118 = 'SOKK-Be'
  640 = 'Sokkolás, max\nPt ellenállás (Ohm):'
  646 = 'Sokkolás, max \nPt ellenállás (Ohm):'
  649 = 'Sokkolás, max \nPt ellenállás [Ohm]:'
  276 = 'SOKK_OK'
  475 = 'SOK_OKK'
  148 = 'Speed1'
  146 = 'SpeedReached'
  91 = 'START'
  258 = 'Start'
  259 = 'Start 1. fázis'
  260 = 'Start 2. fázis'
  879 = 'State'
  75 = 'STOP'
  289 = 'STOP érték'
  98 = 'StromFehler'
  793 = 'STÁTUSZ'
  215 = 'SZERVIZBOXHOZ'
  262 = 'Szervizboxhoz'
  355 = 'Szervíz'
  671 = 'SZERVÍZ'
  626 = 'SZERVÍZBOX'
  633 = 'SZERVÍZBOX / KAMERA'
  548 = 'Szervízbox pozíció'
  632 = 'SZERVÍZBOX/KAMERA'
  315 = 'Szervízboxhoz'
  458 = 'SZERVÍZBOXHOZ'
  371 = 'Szervó hajtás'
  0 = 'Szia'
  472 = 'Szigetelés'
  499 = 'SZIGETELÉS'
  528 = 'Szigetelés érték'
  500 = 'Szigetelési érték (V)'
  652 = 'Szigetelési érték [V]'
  501 = 'SZIG_OK'
  496 = 'Szán pozíció:'
  565 = 'Sürített levegö nyomás'
  571 = 'Sürített levegö nyomás rendben'
  169 = 'TCP'
  874 = 'TCP Close'
  590 = 'TCP IP kapcsolatok törölve'
  873 = 'TCP Open'
  871 = 'TCP Receive'
  875 = 'TCP Send'
  180 = 'TEACH'
  487 = 'Teljes'
  869 = 'Teljes himba\nmüvelet'
  868 = 'Teljes himba müvelet'
  460 = 'Teljes Kappe müvelet'
  461 = 'Teljes kappe müvelet'
  275 = 'Teljes Kappe művelet'
  486 = 'TELJES MÉRÉS'
  696 = 'Teljes/etalon'
  697 = 'Teljes/Etalon'
  52 = 'Tengely'
  408 = 'TENGELY'
  63 = 'Tengely1'
  526 = 'Tengelyek'
  617 = 'Tengelypozíciók'
  51 = 'Tengelíy'
  257 = 'Termelés'
  312 = 'Termelés 1. fázis'
  313 = 'Termelés 2. fázis'
  667 = 'Termék típus'
  664 = 'TERMÉK TÍPUS:'
  666 = 'Terméktípus'
  918 = 'TERMÉKVÁLTÁS'
  248 = 'Ticker'
  310 = 'Tovább'
  281 = 'TÍPUSVÁLASZTÁS'
  5626 = 'Töröl'
  197 = 'U12V'
  119 = 'U48V'
  553 = 'U:'
  110 = 'UISOL'
  511 = 'Ultimate script-ben megírt parancsok pdf-ben'
  720 = 'um'
  131 = 'Utasítás'
  244 = 'Utolsó érték (C)'
  245 = 'Utolsó érték (s)'
  158 = 'Vagashoz'
  151 = 'Vago/hajito'
  19 = 'Valami'
  102 = 'VEGMEROHOZ'
  815 = 'VENTILLÁTOROK1'
  816 = 'VENTILLÁTOROK2'
  271 = 'VENTING'
  915 = 'Vezeték '
  913 = 'Vezeték pozíció'
  607 = 'Vezeték sorrend  OK'
  914 = 'Vezeték szín sorrend'
  343 = 'Vezérlö panel'
  344 = 'Vezérlő panel'
  558 = 'VIGYÁZAT!!! CSAK AKKOR INDÍTSUNK LÉZEREZÉST,\nHA A LÉZERSUGÁR ELZÁRT TÉRBEN MARAD,'
  562 = 'VIGYÁZAT!!! CSAK AKKOR INDÍTSUNK LÉZEREZÉST,\nHA A LÉZERSUGÁR ELZÁRT TÉRBEN MARAD,\nVAGY HA A VESZÉLYEZTETETTEK MEGFELELÖ\nVÉDÖSZEMÜVEGET VISELNEK!\n\nA LÉZER HULLÁMHOSSZA: 1064 nm\nLÉZEROSZTÁLY: 4\nMAX. TELJESÍTMÉNY: 10 W'
  560 = 'VIGYÁZAT!!! CSAK AKKOR INDÍTSUNK LÉZEREZÉST,\nHA A LÉZERSUGÁR ELZÁRT TÉRBEN MARAD,\nVAGY HA A VESZÉLYEZTETETTEK MEGFELELŐ\nVÉDŐSZEMÜVEGET VISELNEK!\n\nA LÉZER HULLÁMHOSSZA: 1064 nm\nLÉZEROSZTÁLY: 4'
  561 = 'VIGYÁZAT!!! CSAK AKKOR INDÍTSUNK LÉZEREZÉST,\nHA A LÉZERSUGÁR ELZÁRT TÉRBEN MARAD,\nVAGY HA A VESZÉLYEZTETETTEK MEGFELELŐ\nVÉDŐSZEMÜVEGET VISELNEK!\n\nA LÉZER HULLÁMHOSSZA: 1064 nm\nLÉZEROSZTÁLY: 4\nMAX. TELJESÍTMÉNY: 10 W'
  559 = 'VIGYÁZAT!!! CSAK AKKOR INDÍTSUNK LÉZEREZÉST,\nHA A LÉZERSUGÁR ELZÁRT TÉRBEN MARAD,\nVAGY HA A VESZÉLYEZTETETTEK MEGFELELŐ\nVÉDŐSZEMÜVEGET VISELNEK!\nA LÉZER HULLÁMHOSSZA: 1064 nm\nLÉZEROSZTÁLY: 4'
  605 = 'Vizsgálat'
  95 = 'Vorwarnung'
  378 = 'Vágáshoz'
  375 = 'Vágó/hajító'
  540 = 'Vákuum A'
  539 = 'Vákuum B'
  535 = 'VÁKUUM BE'
  536 = 'VÁKUUM KI'
  538 = 'VákuumA'
  533 = 'VÁKUUMTAPPANCS FEL'
  534 = 'VÁKUUMTAPPANCS LE'
  8896 = 'Válassza ki a gyártani kívánt terméktípust!\nÜgyeljen rá, hogy a megfelelő NTC és Pt1000\nalkatrészek legyenek betárazva, felhasználva!'
  3674 = 'Válassza ki a gyártani kívánt terméktípust!\nÜgyeljen rá, hogy a megfelelő NTC és Pt1000\nalkatrészek legyenek betárazva, felhasználva!\nHa kell, ezek vonalkódját is be lehet olvastatni.'
  3788 = 'Válasszon felhasználót a módosításhoz / törléshez vagy adjon meg újat!'
  84 = 'VÉGHAJLITASHOZ'
  195 = 'VÉGHAJLÍTÁS'
  518 = 'VÉGHAJLÍTÁSHOZ'
  353 = 'Véghajlító'
  492 = 'VÉGMÉRÖ'
  493 = 'Végmérö'
  636 = 'VÉGMÉRÖ / LÉZER'
  665 = 'Végmérö alapállapotban'
  543 = 'Végmérö kapcsolási rajz'
  494 = 'Végmérö parancs/üzenet:'
  497 = 'Végmérö pozíció:'
  641 = 'VÉGMÉRÖ RESET'
  498 = 'VÉGMÉRÖHÖZ'
  196 = 'Végmérő'
  594 = 'Végmérő alapállapotban'
  542 = 'Végmérő kapcsolási rajz'
  541 = 'Végmérő kapcsolási rajzyitása'
  489 = 'Végmérő parancs/üzenet:'
  609 = 'végállások'
  178 = 'WARNING'
  550 = 'X:'
  551 = 'Y:'
  552 = 'Z:'
  145 = 'ZeroSpeed'
  675 = 'ZÁR'
  155 = 'Zárva'
  836 = 'Zöld gomb'
  843 = 'Zöld gomb: NTC vágás\nPiros gomb: NTC elengedés'
  423 = 'Állapotgép állapota:'
  455 = 'Állapotváltozó: %s'
  524 = 'Állomáshelyek pozíciói:'
  360 = 'ÁRAMHIBA'
  357 = 'ÁRAMMAL'
  580 = 'Árammal hegesztés BE'
  806 = 'ÉLETTARTAM FIGYELÉS'
  334 = 'Értékelés'
  848 = 'ÚJ\nPANEL'
  5620 = 'Új / Módosít'
  290 = 'Új NTC'
  261 = 'ÚJ NTC VÁGÁS'
  474 = 'ÚJ PANEL'
  796 = 'Újra-'
  797 = 'Újra-\nmérés'
  597 = 'ÚJRAINDÍTÁS'
  280 = 'Útmérés'
  361 = 'ÜZEMKÉSZ'
END_TEXTLIST

// ---- POUs/AUTOMATA_lepesek1.TcTLO
TEXTLIST AUTOMATA_lepesek1
  0 = 'Készenléti állapot'
  1 = 'Várakozás az NTC vágóra'
  2 = 'A szán indítása'
  3 = 'A szán az előhajlítóhoz mozog...'
  4 = 'Előhajlítás...'
  5 = 'Véghajlításhoz indul'
  6 = 'A szán a véghajlításhoz mozog...'
  7 = 'Véghajlítás indítása'
  8 = 'Véghajlítás...'
  9 = 'A szán indítása'
  10 = '1. hegesztés, várakozás a szánra'
  11 = '1. hegesztés, fej indítása'
  12 = '1. hegesztés, várakozás a fejre'
  13 = '1. hegesztés folyamatban...'
  14 = '1. hegesztés, fej vissza'
  15 = '1. hegesztés, fej vissza'
  16 = '3. hegesztés, várakozás a szánra'
  17 = '3. hegesztés, fej indítása'
  18 = '3. hegesztés, várakozás a fejre'
  19 = '3. hegesztés, hegesztés folyamatban'
  20 = '3. hegesztés, fej vissza'
  21 = '3. hegesztés, fej vissza'
  22 = '2. hegesztés, várakozás a szánra'
  23 = '2. hegesztés, fej indítása'
  24 = '2. hegesztés, várakozás a fejre'
  25 = '2. hegesztés, hegesztés folyamatban'
  26 = '2. hegesztés, fej vissza'
  27 = '2. hegesztés, fej vissza'
  28 = '4. hegesztés, várakozás a szánra'
  29 = 'Várakozás az NTC vágás végére'
  30 = 'Várakozás a robotra'
  31 = 'A robot az NTC-ért megy'
  32 = 'A robot az NTC-ért megy'
  33 = 'Várakozás az NTC elengedésére'
  34 = 'A robot az NTC-t a 4. hegesztéshez viszi'
  35 = '4. hegesztés, fej indítása'
  36 = '4. hegesztés, várakozás a fejre'
  37 = '4. hegesztés, hegesztés folyamatban'
  38 = '4. hegesztés, fej vissza'
  39 = '4. hegesztés, fej vissza'
  40 = '4. hegesztés, robot elmegy'
  41 = '4. hegesztés, robot elmegy'
  42 = '5. hegesztés, várakozás a szánra'
  43 = '5. hegesztés, fej indítása'
  44 = '5. hegesztés, várakozás a fejre'
  45 = '5. hegesztés, hegesztés folyamatban'
  46 = '5. hegesztés, fej vissza'
  47 = '5. hegesztés, fej vissza'
  48 = 'A szán indítása'
  49 = 'A szán a kamerás ellenörzéshez mozog...'
  50 = 'Kamerás végértékelés'
  60 = 'A szán a kamerás ellenörzéshez mozog...'
  61 = 'Betett termék kamerás ellenörzése'
  62 = 'A szán indítása'
  99 = 'STOP utáni várakozás'
  100 = 'A szán indítása a szervízboxhoz'
  101 = 'Szervízbox, várakozás a szánra'
  102 = 'Várakozás az adapter\nkivételére'
  103 = 'Várakozás az adapter\nkivétele után'
  105 = 'Várakozás...'
  110 = 'NTC vágó ellenörzése'
  111 = 'Döntés új NTC vágásról'
  112 = 'Várakozás az NTC vágóra'
  113 = 'Várakozás az NTC megfogó nyitására'
  120 = 'Termék berakás, megigazítás'
  121 = 'Várakozás a folytatásra'
  130 = 'NTC tengely leállítása'
  131 = 'Hegesztöfejek visszahúzása'
  132 = 'Várakozás a hegesztöfejek\nvisszahúzódására'
  133 = 'Robot pozíció ellenörzése'
  134 = 'Robot HOME-ba érkezésére vár'
  135 = 'Várakozás a hajlító- és\nhegesztöfejek visszahúzódására'
  140 = '1. hegesztöfej visszahúzása'
  141 = 'Várakozás az 1. hegesztőfej\nvisszahúzódására'
  142 = 'Várakozás a szán szervízboxba\n\nérkezésére'
  143 = 'Várakozás a folytatásra'
  150 = '1. hegesztöfej visszahúzása'
  151 = 'Várakozás az 1. hegesztőfej\nvisszahúzódására'
  152 = 'Várakozás a szán szervízboxba\n\nérkezésére'
  153 = 'Várakozás a folytatásra'
  160 = '1. hegesztöfej visszahúzása'
  161 = 'Várakozás az 1. hegesztőfej\nvisszahúzódására'
  162 = 'Várakozás a szán szervízboxba\n\nérkezésére'
  163 = 'Várakozás a folytatásra'
  170 = '2. hegesztöfej visszahúzása'
  171 = 'Várakozás az 2. hegesztőfej\nvisszahúzódására'
  172 = 'Várakozás a folytatásra'
  180 = '2. hegesztöfej visszahúzása'
  181 = 'Várakozás az 2. hegesztőfej\nvisszahúzódására'
  182 = 'Várakozás a szán szervízboxba\n\nérkezésére'
  183 = 'Várakozás a folytatásra'
  190 = 'Adapter pótlólagos felhelyezése, munkadarab rögzítése'
  300 = 'NTC oldali folyamat felfüggesztve'
  200 = 'Adapter vissza kezelőhöz sorja vágás miatt!'
  201 = 'Vegye ki az adaptert és vágja le a sorját!'
  203 = 'Tegye vissza az adaptert sorja vágás után!'
  204 = "Nyomja meg a 'Tovább' gombot!"
   = ''
END_TEXTLIST

// ---- POUs/AUTOMATA_lepesek2.TcTLO
TEXTLIST AUTOMATA_lepesek2
  0 = 'Készenléti állapot'
  1 = 'A szán indítása'
  3 = '6. hegesztés, várakozás a szánra'
  4 = '6. hegesztés, fej indítása'
  5 = '6. hegesztés, várakozás a fejre'
  6 = '6. hegesztés, hegesztés folyamatban'
  7 = '6. hegesztés, fej vissza'
  8 = '6. hegesztés, fej vissza'
  9 = 'A szán indítása'
  11 = '7. hegesztés, várakozás a szánra'
  12 = '7. hegesztés, fej indítása'
  13 = '7. hegesztés, várakozás a fejre'
  14 = '7. hegesztés, hegesztés folyamatban'
  15 = '7. hegesztés, fej vissza'
  16 = '7. hegesztés, fej vissza'
  17 = 'A szán indítása'
  18 = 'Kappe felhelyezés, várakozás a szánra'
  19 = 'Várakozás a robotra'
  20 = 'A robot eredmény törlésére vár'
  21 = 'A robot felhelyezi a kappét'
  22 = 'A szán indítása'
  23 = 'Kappe rögzítés, várakozás a szánra'
  24 = 'Kappe rögzítés indítása'
  27 = 'Várakozás a kappe rögzítés végére'
  28 = 'Mérés, várakozás a szánra'
  29 = 'Mérésválasztás'
  30 = 'Várakozás a mérés végére'
  31 = 'Lézeres jelölés előkészítése'
  32 = 'Várakozás a lézerre'
  33 = 'Lézertakaró nyitása'
  34 = 'Lézeres jelölés folyamatban'
  35 = 'Lézerezés állapot lekérdezés'
  36 = 'Lézerezés állapot lekérdezés'
  37 = 'Lézerezés állapot lekérdezés'
  40 = 'Lézertakaró zárása'
  41 = 'Kódellenörzés, várakozás a szánra'
  42 = 'Kódellenörzés folyamatban'
  43 = 'Kódellenörzés folyamatban'
  60 = 'Kiértékelés'
  99 = 'STOP utáni várakozás'
  100 = 'A szán indítása a szervízboxhoz'
  101 = 'Szervízbox, várakozás a szánra'
  103 = 'Várakozás az adapter\nkivételére'
  104 = 'Várakozás az adapter\nkivétele után'
  105 = 'Hegesztési hiba utáni várakozás'
  110 = 'A szán indítása a szervízboxhoz'
  111 = 'Várakozás a szánra és a folytatásra'
  112 = 'Várakozás a végmérőre, szán indítása'
  120 = 'Adapter pótlólagos felhelyezése'
  130 = 'Elhárítandó lézerhiba'
  140 = 'A szán indítása a szervízboxhoz'
  141 = 'Fedél megigazítására vár'
  142 = 'Kappe felhelyezés, várakozás a szánra'
  143 = 'Kappe felhelyezés indítása'
  150 = 'A szán indítása a szervízboxhoz'
  151 = 'Kappe pótlólagos felrakására vár'
  152 = 'Kappe felhelyezés, várakozás a szánra'
  153 = 'Kappe felhelyezés indítása'
  160 = 'Logolás hiba, várakozás a "Tovább" gombra.'
  170 = 'Várakozás folytatásra'
  171 = 'Hibás termék elengedése'
  180 = 'A szán a szervízboxhoz jön'
  181 = 'A "Tovább" gombra vár'
  200 = 'Pt tengely leállítása'
  201 = 'Hegesztés leállítása'
  202 = 'Hegesztö hibatörlés ellenörzése'
  203 = 'Sikertelen hegesztö hibatörlés\nutáni várakozás'
  204 = 'Várakozás a hegesztöfej\nvisszahúzódására'
  205 = 'Robot pozíció ellenörzése'
  206 = 'Robot HOME-ba érkezésére vár'
  207 = 'Végmérö RESET-elése'
  208 = 'Kappe RESET-elése'
  209 = 'Kappe RESET-elése'
  212 = 'Várakozás a végmérö, a lézer takaró lemez\nés a hegezstöfej alapállapotára'
  300 = 'Pt oldali folyamat felfüggesztve'
  400 = 'Kamera indítás'
  401 = 'Kamera kiértékelés'
  402 = 'Következö engedélyezett\nmüvelethez indul'
  410 = 'Várakozás a szánra ill. a\nfolytatásra'
  190 = 'A szán indítása a szervízboxhoz'
  191 = 'Szervízbox, várakozás a szánra'
  192 = 'A "Tovább" gombra vár'
  500 = 'Csatlakozó érzékeléshez'
  501 = 'Csatlakozó érzékelés indul'
  502 = 'Csatlakozó érzékelés kiértékelés'
  503 = 'A szán indítása'
  210 = 'Himba RESET-elése'
  211 = 'Himba RESET-elése'
   = ''
END_TEXTLIST

// ---- POUs/DUT_types.TcTLO
TEXTLIST DUT_types
  0 = 'Etalon 1'
  1 = 'Etalon 2'
  2 = 'Etalon 3'
  3 = 'Termék'
   = ''
END_TEXTLIST

// ---- POUs/ErrorList.TcTLO
TEXTLIST ErrorList
  0 = 'Minden rendben.'
  1 = 'Termék csatlakozó fedél\nnincs nyitva.'
  2 = 'Termék csatlakozó fedél\nnyitva van.'
  3 = 'Fütötömb hömérséklete\nnem megfelelö.'
  4 = 'Fütötömb hömérséklete\nmegfelelö.'
  5 = 'Sürített levegö nyomása\nnincs rendben.'
  6 = 'Sürített levegö nem kapcsolt ki.'
  7 = 'Nincs hegesztö\nelöfigyelmeztetés.'
  8 = 'Hegesztö\nelöfigyelmeztetés!'
  9 = 'Nem kell hegesztö elektródát\ncserélni.'
  10 = 'Hegesztö elektródát\nkell cserélni.'
  11 = 'A hegesztö még nem\nindult be.'
  12 = 'A hegesztö beindult.'
  13 = 'Nincs hegesztö áramhiba.'
  14 = 'Hegesztö áramhiba!'
  15 = 'Árammal hegesztés\nkikapcsolva!'
  16 = 'Árammal hegesztés\nbekapcsolva!'
  17 = 'A hegesztö nem üzemkész!'
  18 = 'A hegesztö üzemkész!'
  19 = 'NTC vágó: sebesség\nnem nulla.'
  20 = 'NTC vágó: sebesség nulla.'
  21 = 'NTC vágó: a sebesség\nnem állt be!'
  22 = 'NTC vágó: a sebesség\nbeállt!'
  23 = 'NTC vágó: nincs vészjelzés.'
  24 = 'NTC vágó: vészjelzés!'
  25 = 'NTC vágó: nem üzemkész!'
  26 = 'NTC vágó: üzemkész.'
  27 = 'Hegesztö: hegesztési\nfolyamat nincs kész.'
  28 = 'Hegesztö: hegesztési\nfolyamat kész.'
  29 = 'Pt oldali fénysorompó\nblokkolva.'
  30 = 'Pt oldali fénysorompó\nszabad.'
  31 = 'NTC oldali fénysorompó\nblokkolva.'
  32 = 'NTC oldali fénysorompó\nszabad.'
  33 = 'A kamera dolgozik.'
  34 = 'A kamera nem dolgozik.'
  35 = 'Kamera: a termék nincs jól\nrögzitve.'
  36 = 'Kamera: a termék jól\nvan rögzitve.'
  37 = 'Kamera: vezeték színsorrend\nnincs rendben.'
  38 = 'Kamera: vezeték színsorrend\nrendben van.'
  39 = 'Kamera: vezeték szigetelés\nnincs rendben.'
  40 = 'Kamera: vezeték szigetelés\nrendben van.'
  41 = 'A biztonsági relé földje megvan.'
  42 = 'A biztonsági relé földje hiányzik.\nValamelyik ajtó nyitva van?'
  43 = 'A biztonsági relé tápja hiányzik.\nValamelyik ajtó nyitva van?'
  44 = 'A biztonsági relé tápja megvan.'
  65 = 'Adapterlefogó nincs\nteljesen visszahúzva.'
  66 = 'Adapterlefogó\nteljesen visszahúzva.'
  67 = 'Adapterlefogó nem\naktiválódott.'
  68 = 'Az adapterlefogó aktív.'
  69 = 'Nem érzékel adaptert\na szánon!'
  70 = 'Fent van az adapter a szánon.'
  71 = 'A 3-as hegesztöfej nincs fent.'
  72 = 'A 3-as hegesztöfej fent van.'
  73 = 'A 3-as hegesztöfej nincs lent.'
  74 = 'A 3-as hegesztöfej lent van.'
  75 = 'A Pt oldali tengely plusz\nvégállásban van.'
  76 = 'A Pt oldali tengely nincs\nplusz \nvégállásban.'
  81 = 'Fütötömb nincs fent.'
  82 = 'Fütötömb fent van.'
  83 = 'Fütötömb nincs lent.'
  84 = 'Fütötömb lent van.'
  85 = 'Mérötük nincsenek kitolva.'
  86 = 'Mérötük ki vannak tolva.'
  87 = 'Mérötük nincsenek behúzva.'
  88 = 'Mérötük be vannak húzva.'
  89 = 'Lézer blende nincs bezárva.'
  90 = 'Lézer blende be van zárva.'
  91 = 'Lézer blende nincs kinyitva.'
  92 = 'Lézer blende ki van nyitva.'
  93 = 'Kappe prés legalul van.'
  94 = 'Kappe prés nincs legalul.'
  95 = 'A Pt oldali tengely minusz\nvégállásban van.'
  96 = 'A Pt oldali tengely nincs\nminusz \nvégállásban.'
  97 = 'Kappe prés jobb oldala\nnincs lent.'
  98 = 'Kappe prés jobb oldala\nlent van.'
  99 = 'Kappe prés jobb oldala\nnincs fent.'
  100 = 'Kappe prés jobb oldala\nfent van.'
  101 = 'Kappe prés bal oldala\nnincs fent.'
  102 = 'Kappe prés bal oldala\nfent van.'
  103 = 'Kappe prés bal oldala\nnincs lent.'
  104 = 'Kappe prés bal oldala\nlent van.'
  105 = 'A fütötömb nincs a szán\nfölött.'
  106 = 'A fütötömb a szán \nfölött van.'
  107 = 'A szigetelés mérötük\nnincsenek a szán fölött.'
  108 = 'A szigetelés mérötük\na szán fölött vannak.'
  109 = 'A kappe prés nincs fent.'
  110 = 'A kappe prés fent van.'
  111 = 'A nagyfeszültségü mérötü\nnincs lent.'
  112 = 'A nagyfeszültségü mérötü\nlent van.'
  113 = 'NTC vágó: vágó-hajlító\nnincs lent.'
  114 = 'NTC vágó: vágó-hajlító\nlent van.'
  115 = 'NTC vágó: vágó-hajlító\nnincs fent.'
  116 = 'NTC vágó: vágó-hajlító\nfent van.'
  117 = '2. hegesztö fej: Felsö elektróda\nnincs kitolva.'
  118 = '2. hegesztö fej: Felsö elektróda\nki van tolva.'
  119 = '2. hegesztö fej: Felsö elektróda\nnincs behúzva.'
  120 = '2. hegesztö fej: Felsö elektróda\nbe van húzva.'
  121 = '2. hegesztö fej: Alsó elektróda\nnincs behúzva.'
  122 = '2. hegesztö fej: Alsó elektróda\nbe van húzva.'
  123 = '2. hegesztö fej: Alsó elektróda\nnincs kitolva.'
  124 = '2. hegesztö fej: Alsó elektróda\nki van tolva.'
  125 = 'NTC oldali tengely minusz\nvégállásban van.'
  126 = 'NTC oldali tengely nincs\nminusz \nvégállásban.'
  127 = 'NTC vágó: az NTC nincs\nmegfelelö pozícióban.'
  128 = 'NTC vágó: az NTC\nmegfelelö pozícióban van.'
  129 = 'NTC vágó: NTC megfogó\nnincs nyitva.'
  130 = 'NTC vágó: NTC megfogó\nnyitva van.'
  131 = 'NTC vágó: NTC megfogó\nnincs zárva.'
  132 = 'NTC vágó: NTC megfogó\nzárva van.'
  133 = 'NTC vágó: NTC kiszedö\nnincs kitolva.'
  134 = 'NTC vágó: NTC kiszedö\nki van tolva.'
  135 = 'NTC vágó: NTC kiszedö\nnincs behúzva.'
  136 = 'NTC vágó: NTC kiszedö\nbe van húzva.'
  137 = 'NTC vágó: piros gomb\nnincs benyomva.'
  138 = 'NTC vágó: piros gomb\nbe van nyomva.'
  139 = 'NTC vágó: zöld gomb\nnincs benyomva.'
  140 = 'NTC vágó: zöld gomb\nbe van nyomva.'
  141 = 'Nincs megfelelö vágott NTC.'
  142 = 'Van vágott NTC.'
  145 = 'Elöhajlító: felsö pofa nincs lent.'
  146 = 'Elöhajlító: felsö pofa lent van.'
  147 = 'Elöhajlító: felsö pofa nincs fent.'
  148 = 'Elöhajlító: felsö pofa fent van.'
  149 = 'Elöhajlító: alsó pofa nincs lent.'
  150 = 'Elöhajlító: alsó pofa lent van.'
  151 = 'Elöhajlító: alsó pofa nincs fent.'
  152 = 'Elöhajlító: alsó pofa fent van.'
  153 = '1. hegesztöfej: bal elektróda\nnincs fent.'
  154 = '1. hegesztöfej: bal elektróda\nfent van.'
  155 = '1. hegesztöfej: bal elektróda\nnincs lent.'
  156 = '1. hegesztöfej: bal elektróda\nlent van.'
  161 = 'Véghajlító: felsö pofa nincs lent.'
  162 = 'Véghajlító: felsö pofa lent van.'
  163 = 'Véghajlító: felsö pofa nincs fent.'
  164 = 'Véghajlító: felsö pofa fent van.'
  165 = 'Véghajlító: alsó pofa nincs fent.'
  166 = 'Véghajlító: alsó pofa fent van.'
  167 = 'Véghajlító: alsó pofa nincs lent.'
  168 = 'Elöhajlító: alsó pofa lent van.'
  169 = '1. hegesztöfej: jobb elektróda\nnincs fent.'
  170 = '1. hegesztöfej: jobb elektróda\nfent van.'
  171 = '1. hegesztöfej: jobb elektróda\nnincs lent.'
  172 = '1. hegesztöfej: jobb elektróda\nlent van.'
  175 = 'NTC oldali tengely plusz\nvégállásban van.'
  176 = 'NTC oldali tengely nincs\nplusz végállásban.'
  193 = 'NTC oldali tengely nem\nüzemkész.'
  194 = 'NTC oldali tengely\nüzemkész.'
  195 = 'Pt oldali tengely nem\nüzemkész.'
  196 = 'Pt oldali tengely\nüzemkész.'
  197 = 'Nem kapcsolt be a\nnagyfeszültség.'
  198 = 'Nem kapcsolt ki a\nnagyfeszültség.'
  199 = 'Nincs a \nnagyfeszültség\na kappén.'
  200 = 'Rajta van a nagyfeszültség\na kappén.'
  201 = 'Nincs 48V a sokkoláshoz.'
  202 = 'Van 48V a sokkoláshoz.'
  203 = 'Nem kapcsolt ki a\nnagyfeszültség'
  204 = 'Kikapcsolt a nagyfeszültség.'
  205 = 'A Kappe prés nincs fent.'
  300 = 'NTC vágó állapothiba.'
  301 = 'NTC nem érkezett meg a\nvágáshoz.'
  302 = 'A robot a szán útjában lehet.'
  303 = 'A hegesztöt lefoglalta az\nNTC oldal.'
  304 = 'A hegesztöt lefoglalta a\nPt oldal.'
  305 = 'A robotot lefoglalta az\nNTC oldal.'
  306 = 'A robotot lefoglalta a\nPt oldal.'
  307 = 'A robotmüvelet elakadt.'
  308 = 'Kameramüvelet elakadt.'
  309 = 'Igazítsa meg/tegye fel a Pt pozícionáló\nfedelet, majd nyomja meg a\n"Tovább" gombot!'
  310 = 'Helyezzen be a helyére egy kappét,\nmajd nyomja meg a "Tovább" gombot!'
  311 = 'Nem sikerült a log fájlt\n megnyitni,\nvagy a mappáját létrehozni.'
  312 = 'Nem sikerült lekérdezni a\nlog fájl tulajdonságait.'
  313 = 'Nem sikerült a rendszeridöt\nlekérdezni.'
  314 = 'Nem sikerült írni a log fájlt.'
  315 = 'Nem sikerült a log fájl zárása.'
  316 = 'Nem sikerült létrehozni a log\nfájlnak a megfelelö mappát.'
  317 = 'Nincs lezárva a csatlakozó fedél.\nZárja le és nyomja meg a "Tovább"\ngombot!'
  318 = 'Hibás termék! Nyomja meg a\n"Tovább" gombot, és tegye a \nterméket a megfelelö helyre!'
  319 = 'Termékrögzítés, vezetéksorrend,\nhüvelyek rendben vannak?\nHa igen, nyomja meg a "Tovább" gombot!'
  320 = '1. hegesztés: alkatrész felismerési hiba!'
  321 = '3. hegesztés: alkatrész felismerési hiba!'
  322 = '2. hegesztés: alkatrész felismerési hiba!'
  323 = '4. hegesztés: alkatrész felismerési hiba!'
  324 = '5. hegesztés: alkatrész felismerési hiba!'
  325 = '1. hegesztés: a hegesztés nem megfelelő!'
  326 = '3. hegesztés: a hegesztés nem megfelelő!'
  327 = '2. hegesztés: a hegesztés nem megfelelő!'
  328 = '4. hegesztés: a hegesztés nem megfelelő!'
  329 = '5. hegesztés: a hegesztés nem megfelelő!'
  330 = '1. hegesztés: hegesztési hibát \njelzett a hegesztö'
  331 = '3. hegesztés: hegesztési hibát \njelzett a hegesztö'
  332 = '2. hegesztés: hegesztési hibát \njelzett a hegesztö'
  333 = '4. hegesztés: hegesztési hibát \njelzett a hegesztö'
  334 = '5. hegesztés: hegesztési hibát \njelzett a hegesztö'
  335 = '6. hegesztés: hegesztési hibát \njelzett a hegesztö'
  336 = '7. hegesztés: hegesztési hibát \njelzett a hegesztö'
  337 = 'Ellenörizze a hegesztést, vegye le\na Pt pozícionáló fedelet, majd nyomja\nmeg a "Tovább" gombot!'
  338 = 'Himba nincs elöl'
  339 = 'Himba nincs hátul'
  340 = 'Pt Kamera komm. kapcsolat nyitási hiba!'
  341 = 'Pt Kamera komm. küldési hiba!'
  342 = 'Pt Kamera komm. fogadási hiba!'
  343 = 'Pt Kamera komm. kapcsolat bezárási hiba!'
  344 = 'Pt Kamera nem érzékel terméket!'
  345 = 'Pt Kamera nem érzékel se adaptert, se kappét!\nEllenőrizze a terméket!'
  346 = 'Nincs kiválasztva művelet!'
  347 = 'Pt Kamera adat üres!'
  348 = 'Pt Kamera trigger TimeOut!'
  299 = 'Nincs NTC a hegesztésnél!'
  298 = 'Robot nem OK! Nyissa ki, zárja be a biztonsági ajtót!'
  297 = 'NTC érzékelő hiba!'
  296 = 'Nincs NTC a hegesztésnél!'
  295 = 'Elektródacsere szükséges!'
   = ''
END_TEXTLIST

// ---- POUs/ErrorList1.TcTLO
TEXTLIST ErrorList1
  1 = 'Az NTC vágó foglalt!'
  3 = 'A hajlítók nem állnak készen, vagy nem érkezett meg a szán az előhajlításhoz.'
  4 = 'Nem végzett idöben az elöhajlító.'
  6 = 'Nem érkezett meg a szán a véghajlításhoz.'
  7 = 'Nem állnak készen a hajlítók.'
  8 = 'Nem végzett a véghajlító.'
  10 = 'Nem érkezett meg a szán az első hegesztéshez.'
  12 = 'Nem érkezett meg az 1. hegesztésnél a fej.'
  13 = 'Nem lett kész az 1. hegesztési folyamat.'
  15 = 'Nem húzódott vissza az 1. hegesztésnél a fej.'
  16 = 'Nem érkezett meg a szán a 3. hegesztéshez.'
  18 = 'Nem érkezett meg a 3. hegesztésnél a fej.'
  19 = 'Nem lett kész a 3. hegesztési folyamat.'
  21 = 'Nem húzódott vissza a 3. hegesztésnél a fej.'
  22 = 'Nem érkezett meg a szán a 2. hegesztéshez.'
  24 = 'Nem érkezett meg a 2. hegesztésnél a fej.'
  25 = 'Nem lett kész a 2. hegesztési folyamat.'
  27 = 'Nem húzódott vissza a 2. hegesztésnél a fej.'
  28 = 'Nem érkezett meg a szán a 4. hegesztéshez.'
  29 = 'Nem fejeződött be az NTC vágás.'
  32 = 'Nem áll rendelkezésre a robot vagy nincs levágva az NTC.'
  33 = 'A megfogó nem engedte el a levágott NTC-t.'
  34 = 'A robot még nem vitte oda az NTC-t a hegesztéshez, vagy foglalt a hegesztő.'
  36 = 'Nem érkezett meg a 4. hegesztésnél a fej.'
  37 = 'Nem lett kész a 4. hegesztési folyamat.'
  39 = 'Nem húzódott vissza a 4. hegesztésnél a fej.'
  41 = 'A robot még nem jött el a hegesztés helyétől.'
  42 = 'Nem érkezett meg a szán az 5. hegesztéshez.'
  44 = 'Nem érkezett meg az 5. hegesztésnél a fej.'
  45 = 'Nem lett kész az 5. hegesztési folyamat.'
  47 = 'Nem húzódott vissza az 5. hegesztésnél a fej.'
  110 = 'Nem fejeződött be az NTC vágás.'
  112 = 'Az NTC vágó foglalt.'
  113 = 'Nem fejeződött be az NTC vágás.'
   = ''
END_TEXTLIST

// ---- POUs/ErrorList2.TcTLO
TEXTLIST ErrorList2
  3 = 'Nem érkezett meg a szán a 6. hegesztéshez, vagy foglalt a hegesztő.'
  5 = 'Nem érkezett meg a 6. hegesztésnél a fej.'
  6 = 'Nem lett kész a 6. hegesztési folyamat.'
  8 = 'Nem húzódott vissza a 6. hegesztésnél a fej.'
  11 = 'Nem érkezett meg a szán a 7. hegesztéshez.'
  13 = 'Nem érkezett meg a 7. hegesztésnél a fej.'
  14 = 'Nem lett kész a 7. hegesztési folyamat.'
  16 = 'Nem húzódott vissza a 7. hegesztésnél a fej.'
  18 = 'Nem érkezett meg a szán a Kappe robotművelethez.'
  19 = 'A robot foglalt.'
  20 = 'A robot nem végzett a Kappe felrakásával.'
  22 = 'Nem érkezett meg a szán a kappézáshoz.'
  27 = 'Nem fejeződött be a kappézás művelete.'
  28 = 'Nem érkezett meg a szán a méréshez.'
  30 = 'Nem fejeződött be a mérés.'
  32 = 'Nem sikerült elküldeni a terméktípust a lézernek.'
  33 = 'Nem nyílt ki a lézer takaró.'
  34 = 'Nem sikerült elküldeni a lézernek a lézerezés parancsot.'
  36 = 'Nem záródott be a lézer takaró.'
  37 = 'Nem érkezett meg a szán a kódellenőrzéshez.'
  101 = 'Nem érkezett meg a szán a szervízboxhoz.'
  111 = 'Nem érkezett meg a szán a szervízboxhoz.'
  112 = 'Nem sikerült törölni a végmérő hibaállapotát.'
   = ''
END_TEXTLIST

// ---- VISUs/AddDelete.TcVIS
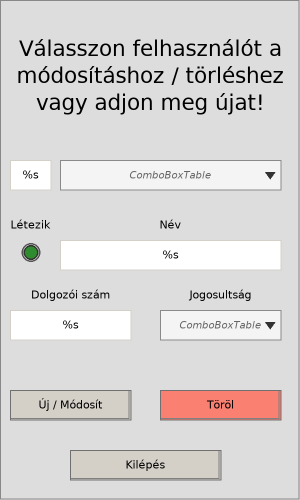
VISUALIZATION AddDelete  // 300x500
    Label (10,10 281x131), "Válasszon felhasználót a módosításhoz / törléshez vagy adjon meg újat!"
    Button (70,450 151x30), "Kilépés"
        toggle GVL.AddDeleteEnabled
    ComboBoxTable (60,160 221x30), variable: GVL.UserID_Temp, data array: GVL.Users
        p3854506369: GVL.Users[INDEX].UserID
        p1892666644: GVL.Users[INDEX].UserNumber
        p338671338: GVL.Users[INDEX].UserName
        p2170511999: GVL.Users[INDEX].UserLevel
        p3723444502: GVL.Users[INDEX].UserExist
    Textfield (10,310 121x30), "%s", text variable: GVL.UserTemp.UserNumber
        OnMouseClick: write the text variable via VisuDialogs.Numpad
    Textfield (60,240 221x30), "%s", text variable: GVL.UserTemp.UserName
        OnMouseClick: write the text variable via Edit
    Button (10,390 121x30), "Új / Módosít"
        toggle GVL.UserModify
    Button (160,390 121x30), "Töröl"
        OnMouseClick: OpenDialog Dialog=Biztos, OpenModal=True, OpenCentered=True
    Label (60,210 221x30), "Név"
    Label (10,280 121x30), "Dolgozói szám"
    Label (160,280 121x30), "Jogosultság"
    Textfield (10,160 41x30), "%s", text variable: GVL.UserTemp.UserID
    Lamp1 (20,240 22x25), variable: GVL.UserTemp.UserExist, style: Lamp-Lamp1-Green
    ComboBoxTable (160,310 121x30), variable: GVL.UserTemp.UserLevel, data array: GVL.UserLevels
        p3854506369: GVL.UserLevels[INDEX]
    Label (10,210 41x30), "Létezik"
END_VISUALIZATION

// ---- VISUs/Biztos.TcVIS
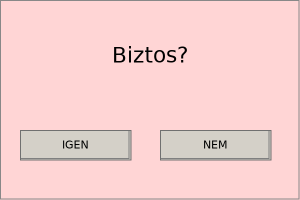
VISUALIZATION Biztos  // 300x200
    Label (10,40 281x30), "Biztos?"
    Button (20,130 111x30), "IGEN"
        toggle GVL.Biztos
        OnMouseClick: CloseDialog Dialog=Biztos, Result=OK, NumpadKeypadSet=True
    Button (160,130 111x30), "NEM"
        OnMouseClick: CloseDialog Dialog=Biztos, Result=OK, NumpadKeypadSet=True
END_VISUALIZATION

// ---- VISUs/Hegesztes_Karbantartas.TcVIS
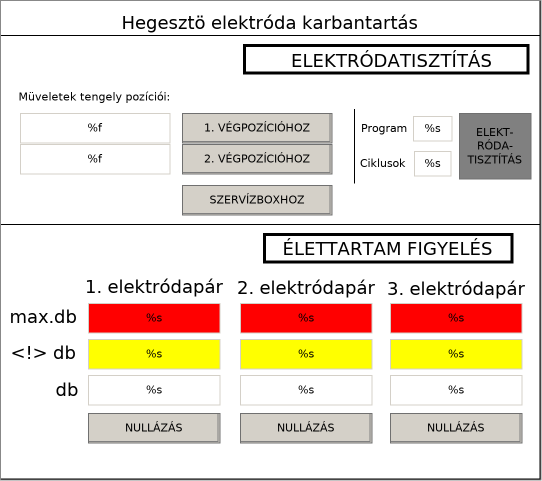
VISUALIZATION Hegesztes_Karbantartas  // 542x481
    Rectangle (0,-1 540x480)
    Textfield (20,113 150x30), "%f", text variable: GVL.lrCsiszoloPosition1
        OnMouseClick: write the text variable via VisuDialogs.Numpad, min -10000, max -1
    Button (182,113 150x30), "1. VÉGPOZÍCIÓHOZ"
        OnMouseUp: execute { JOZSITENGELY.lrJozsiPosition:=GVL.lrCsiszoloPosition1; JOZSITENGELY.sJozsiAxisCommand:='MOVE'; }
    Textfield (20,144 150x30), "%f", text variable: GVL.lrCsiszoloPosition2
        OnMouseClick: write the text variable via VisuDialogs.Numpad, min -10000, max -1
    Button (182,144 150x30), "2. VÉGPOZÍCIÓHOZ"
        OnMouseUp: execute { JOZSITENGELY.lrJozsiPosition:=GVL.lrCsiszoloPosition2; JOZSITENGELY.sJozsiAxisCommand:='MOVE'; }
    Textfield (88,303 132x30), "%s", text variable: GVL.nElectrode1UsageMax
        OnMouseClick: write the text variable via VisuDialogs.Numpad, min 1, max 100000
    Button (88,413 132x30), "NULLÁZÁS"
        OnMouseUp: execute { GVL.nElectrode1Usage:=0; }
    Button (182,185 150x30), "SZERVÍZBOXHOZ"
        OnMouseUp: execute { JOZSITENGELY.lrJozsiPosition:=GVL.lrNTCSzervizbox; JOZSITENGELY.sJozsiAxisCommand:='MOVE'; }
    Button (459,113 72x66), "ELEKT- RÓDA- TISZTÍTÁS"
        OnMouseUp: execute {
            IF GVL.bJOZSITENGELYReserved=FALSE THEN
            	HEGESZTOFEJTISZTITAS.iState:=1;
            END_IF;
        }
    Line (0,35) (540,35), "Hegesztö elektróda karbantartás"
    Line (0,224) (540,224)
    RoundedRectangle (263,233 250x30)
    Label (255,234 265x30), "ÉLETTARTAM FIGYELÉS"
    Label (13,82 163x30), "Müveletek tengely pozíciói:"
    Textfield (413,116 39x25), "%s", text variable: GVL.nHegFejTisztProgram
        OnMouseClick: write the text variable via VisuDialogs.Numpad, min 11, max 14
    Textfield (414,151 37x25), "%s", text variable: GVL.nHegFejTisztCiklusok
        OnMouseClick: write the text variable via VisuDialogs.Numpad, min 1, max 20
    Label (358,116 54x25), "Program"
    Label (357,151 54x25), "Ciklusok"
    Line (354,109) (354,183)
    RoundedRectangle (243,44 286x30)
    Label (255,46 273x30), "ELEKTRÓDATISZTÍTÁS"
    Label (81,272 146x30), "1. elektródapár"
    Label (233,273 146x30), "2. elektródapár"
    Label (383,274 146x30), "3. elektródapár"
    Textfield (88,375 132x30), "%s", text variable: GVL.nElectrode1Usage, colour toggle: GVL.nElectrode1Usage>GVL.nElectrode1UsageWarn
        p2167032090: GVL.nElectrode1AlarmColor
    Textfield (240,303 132x30), "%s", text variable: GVL.nElectrode2UsageMax
        OnMouseClick: write the text variable via VisuDialogs.Numpad, min 1, max 100000
    Button (240,413 132x30), "NULLÁZÁS"
        OnMouseUp: execute { GVL.nElectrode2Usage:=0; }
    Textfield (240,375 132x30), "%s", text variable: GVL.nElectrode2Usage, colour toggle: GVL.nElectrode2Usage>GVL.nElectrode2UsageWarn
        p2167032090: GVL.nElectrode2AlarmColor
    Textfield (390,303 132x30), "%s", text variable: GVL.nElectrode3UsageMax
        OnMouseClick: write the text variable via VisuDialogs.Numpad, min 1, max 100000
    Button (390,413 132x30), "NULLÁZÁS"
        OnMouseUp: execute { GVL.nElectrode3Usage:=0; }
    Textfield (390,375 132x30), "%s", text variable: GVL.nElectrode3Usage, colour toggle: GVL.nElectrode3Usage>GVL.nElectrode3UsageWarn
        p2167032090: GVL.nElectrode3AlarmColor
    Label (5,302 77x30), "max.db"
    Label (52,375 30x30), "db"
    Label (5,338 77x30), "<!> db"
    Textfield (88,339 132x30), "%s", text variable: GVL.nElectrode1UsageWarn
        OnMouseClick: write the text variable via VisuDialogs.Numpad, min 1, max 100000
    Textfield (240,339 132x30), "%s", text variable: GVL.nElectrode2UsageWarn
        OnMouseClick: write the text variable via VisuDialogs.Numpad, min 1, max 100000
    Textfield (390,339 132x30), "%s", text variable: GVL.nElectrode3UsageWarn
        OnMouseClick: write the text variable via VisuDialogs.Numpad, min 1, max 100000
END_VISUALIZATION

// ---- VISUs/Hegesztofej_IOk.TcVIS
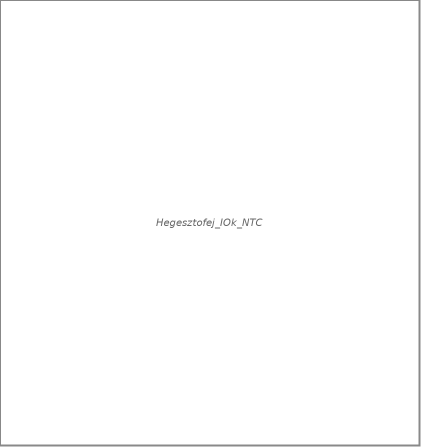
VISUALIZATION Hegesztofej_IOk  // 421x447
    TabControl (0,0 419x445), frame switch variable: GVL.iTengelyLapozo
        shows Hegesztofej_IOk_NTC()
        shows Hegesztofej_IOk_Pt()
        [0]: TabTitle=NTC oldal
        [1]: TabTitle=Pt oldal
END_VISUALIZATION

// ---- VISUs/Hegesztofej_IOk_Pt.TcVIS
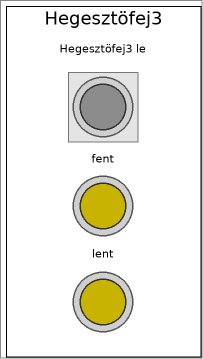
VISUALIZATION Hegesztofej_IOk_Pt  // 203x359
    Rectangle (6,6 195x351), "Hegesztöfej3"
    Lamp1 (68,171 70x70), variable: GVL.bHegeszto3Fent, style: Lamp-Lamp1-Yellow
    Label (73,149 60x20), "fent"
    Lamp1 (68,267 70x70), variable: GVL.bHegeszto3Lent, style: Lamp-Lamp1-Yellow
    Label (73,244 60x20), "lent"
    Label (45,39 116x20), "Hegesztöfej3 le"
    PushSwitch (68,72 70x70), variable: HEGESZTOK.bHegesztoFejekOutput[2], behaviour: TOGGLE, style: Switch-PushSwitch-Gray
END_VISUALIZATION

// ---- VISUs/Hegesztofej_IOk_NTC.TcVIS
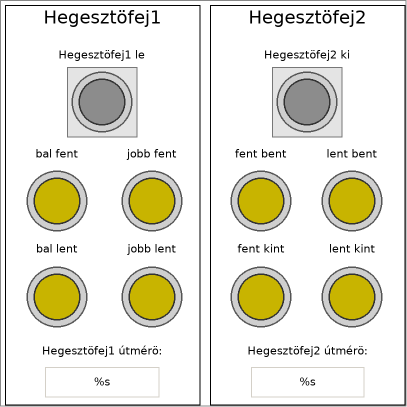
VISUALIZATION Hegesztofej_IOk_NTC  // 407x407
    Group (5,5 195x400)
        Rectangle (0,0 195x400), "Hegesztöfej1"
        Textfield (40,362 114x30), "%s", text variable: HEGESZTOK.ulHegeszto1Utmero, input disabled if: TRUE
        Label (34,336 126x20), "Hegesztöfej1 útmérö:"
        Lamp1 (17,161 70x70), variable: GVL.bHegeszto1BalFent, style: Lamp-Lamp1-Yellow
        Label (22,139 60x20), "bal fent"
        Lamp1 (17,257 70x70), variable: GVL.bHegeszto1BalLent, style: Lamp-Lamp1-Yellow
        Label (22,234 60x20), "bal lent"
        Lamp1 (112,161 70x70), variable: GVL.bHegeszto1JobbFent, style: Lamp-Lamp1-Yellow
        Label (117,139 60x20), "jobb fent"
        Lamp1 (112,257 70x70), variable: GVL.bHegeszto1JobbLent, style: Lamp-Lamp1-Yellow
        Label (117,234 60x20), "jobb lent"
        PushSwitch (62,62 70x70), variable: HEGESZTOK.bHegesztoFejekOutput[0], behaviour: TOGGLE, style: Switch-PushSwitch-Gray
        Label (39,40 116x20), "Hegesztöfej1 le"
    Group (210,5 195x400)
        Rectangle (0,0 195x400), "Hegesztöfej2"
        Textfield (41,362 113x30), "%s", text variable: HEGESZTOK.ulHegeszto2Utmero, input disabled if: TRUE
        Label (33,336 129x20), "Hegesztöfej2 útmérö:"
        Lamp1 (16,257 70x70), variable: GVL.bHegeszto2FentKint, style: Lamp-Lamp1-Yellow
        Label (21,234 60x20), "fent kint"
        Lamp1 (16,161 70x70), variable: GVL.bHegeszto2FentBent, style: Lamp-Lamp1-Yellow
        Label (21,139 60x20), "fent bent"
        Lamp1 (107,257 70x70), variable: GVL.bHegeszto2LentKint, style: Lamp-Lamp1-Yellow
        Label (112,234 60x20), "lent kint"
        Lamp1 (107,161 70x70), variable: GVL.bHegeszto2LentBent, style: Lamp-Lamp1-Yellow
        Label (112,139 60x20), "lent bent"
        Label (39,40 116x20), "Hegesztöfej2 ki"
        PushSwitch (62,62 70x70), variable: HEGESZTOK.bHegesztoFejekOutput[1], behaviour: TOGGLE, style: Switch-PushSwitch-Gray
END_VISUALIZATION

// ---- VISUs/Himba.TcVIS
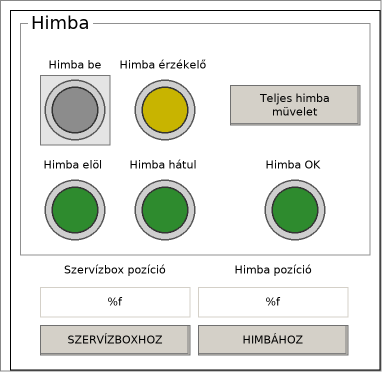
VISUALIZATION Himba  // 382x372
    Rectangle (10,10 370x360)
    GroupBox (20,15 350x240), "Himba"
        PushSwitch (20,60 70x70), variable: HIMBA.bHimba, behaviour: TOGGLE, style: Switch-PushSwitch-Gray
        Label (20,40 70x20), "Himba be"
        Group (0,140 106x90)
            Label (0,0 106x20), "Himba elöl"
            Lamp1 (20,20 70x70), variable: HIMBA.bHimba_elol, style: Lamp-Lamp1-Green
        Group (90,40 106x90)
            Lamp1 (20,20 70x70), variable: HIMBA.bHimba_szenzor, invisible if: GVL.bPtKameraTrigger OR GVL.bPtKameraHegesztesOK, style: Lamp-Lamp1-Yellow
            Label (0,0 106x20), "Himba érzékelő"
        Group (90,140 106x90)
            Lamp1 (20,20 70x70), variable: HIMBA.bHimba_hatul, style: Lamp-Lamp1-Green
            Label (0,0 106x20), "Himba hátul"
        Group (220,140 106x90)
            Lamp1 (20,20 70x70), variable: GVL.bHimbaOK, style: Lamp-Lamp1-Green
            Label (0,0 106x20), "Himba OK"
        Button (210,70 130x40), "Teljes himba müvelet", input disabled if: HIMBA.bHimba_elol=HIMBA.bHimba_hatul
            OnMouseUp: execute { HIMBA.s_InCommand:='START'; }
    Textfield (40,287 150x30), "%f", text variable: GVL.lrPtSzervizbox
    Button (40,325 150x30), "SZERVÍZBOXHOZ"
        OnMouseUp: execute { PISTITENGELY.lrPistiPosition:=GVL.lrPtSzervizbox; PISTITENGELY.sPistiAxisCommand:='MOVE'; }
    Label (40,260 150x20), "Szervízbox pozíció"
    Textfield (198,287 150x30), "%f", text variable: GVL.lrPtKameraPosition
        OnMouseClick: write the text variable via VisuDialogs.Numpad, min -10000, max -1
    Button (198,325 150x30), "HIMBÁHOZ"
        OnMouseUp: execute { PISTITENGELY.lrPistiPosition:=GVL.lrHegesztoPosition6; PISTITENGELY.sPistiAxisCommand:='MOVE'; }
    Label (198,260 150x20), "Himba pozíció"
END_VISUALIZATION

// ---- VISUs/Kamera_Pt.TcVIS
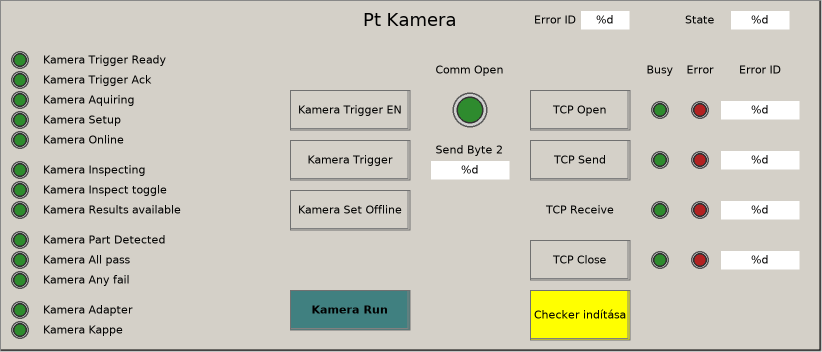
VISUALIZATION Kamera_Pt  // 822x352
    Rectangle (0,0 820x350)
    Lamp1 (450,90 40x40), variable: KAMERAREMOTE.bKameraCommOpen, style: Lamp-Lamp1-Green
    Label (530,200 100x20), "TCP Receive"
    Lamp1 (650,100 20x20), variable: KAMERAREMOTE.bConnectBusy, style: Lamp-Lamp1-Green
    Label (350,0 120x40), "Pt Kamera"
    Button (530,90 100x40), "TCP Open"
        tap KAMERAREMOTE.bKameraCommOpenEnable p1329445385=TRUE
    Button (530,240 100x40), "TCP Close"
        tap KAMERAREMOTE.bKameraCommCloseEnable
    Button (530,140 100x40), "TCP Send"
        tap KAMERAREMOTE.bKameraCommandSend
    Lamp1 (690,100 20x20), variable: KAMERAREMOTE.bConnectError, style: Lamp-Lamp1-Red
    Label (640,60 40x20), "Busy"
    Label (680,60 40x20), "Error"
    Textfield (720,100 80x20), "%d", text variable: KAMERAREMOTE.nConnectErrId
    Label (730,60 60x20), "Error ID"
    Lamp1 (650,250 20x20), variable: KAMERAREMOTE.bCloseBusy, style: Lamp-Lamp1-Green
    Lamp1 (690,250 20x20), variable: KAMERAREMOTE.bCloseError, style: Lamp-Lamp1-Red
    Textfield (720,250 80x20), "%d", text variable: KAMERAREMOTE.nCloseErrId
    Lamp1 (650,150 20x20), variable: KAMERAREMOTE.bSendBusy, style: Lamp-Lamp1-Green
    Lamp1 (690,150 20x20), variable: KAMERAREMOTE.bSendError, style: Lamp-Lamp1-Red
    Textfield (720,150 80x20), "%d", text variable: KAMERAREMOTE.nSendErrId
    Lamp1 (650,200 20x20), variable: KAMERAREMOTE.bReceiveBusy, style: Lamp-Lamp1-Green
    Lamp1 (690,200 20x20), variable: KAMERAREMOTE.bReceiveError, style: Lamp-Lamp1-Red
    Textfield (720,200 80x20), "%d", text variable: KAMERAREMOTE.nReceiveErrId
    Label (430,60 79x20), "Comm Open"
    Label (680,10 40x20), "State"
    Textfield (730,10 60x20), "%d", text variable: KAMERAREMOTE.iState
    Button (290,90 120x40), "Kamera Trigger EN"
        toggle KAMERAREMOTE.bKameraTriggerEN
    Button (290,140 120x40), "Kamera Trigger"
        toggle AUTOMATA.bKameraTrig
    Button (290,190 120x40), "Kamera Set Offline"
        toggle KAMERAREMOTE.bKameraSetOffline
    Textfield (430,160 80x20), "%d", text variable: KAMERAREMOTE.baSendByteArray[2]
    Label (430,140 79x20), "Send Byte 2"
    Label (530,10 50x20), "Error ID"
    Textfield (580,10 50x20), "%d", text variable: KameraProcess.n_OutErrId
    Lamp1 (10,50 20x20), variable: KAMERAREMOTE.bKameraTriggerReady, style: Lamp-Lamp1-Green
    Label (40,50 210x20), "Kamera Trigger Ready"
    Lamp1 (10,70 20x20), variable: KAMERAREMOTE.bKameraTriggerAck, style: Lamp-Lamp1-Green
    Label (40,70 210x20), "Kamera Trigger Ack"
    Lamp1 (10,90 20x20), variable: KAMERAREMOTE.bKameraAcquiring, style: Lamp-Lamp1-Green
    Label (40,90 210x20), "Kamera Aquiring"
    Lamp1 (10,110 20x20), variable: KAMERAREMOTE.bKameraSetup, style: Lamp-Lamp1-Green
    Label (40,110 210x20), "Kamera Setup"
    Lamp1 (10,130 20x20), variable: KAMERAREMOTE.bKameraOnline, style: Lamp-Lamp1-Green
    Label (40,130 210x20), "Kamera Online"
    Lamp1 (10,160 20x20), variable: KAMERAREMOTE.bKameraInspecting, style: Lamp-Lamp1-Green
    Label (40,160 210x20), "Kamera Inspecting"
    Lamp1 (10,180 20x20), variable: KAMERAREMOTE.bKameraInspectToggle, style: Lamp-Lamp1-Green
    Label (40,180 210x20), "Kamera Inspect toggle"
    Lamp1 (10,200 20x20), variable: KAMERAREMOTE.bKameraResultsAvble, style: Lamp-Lamp1-Green
    Label (40,200 210x20), "Kamera Results available"
    Lamp1 (10,230 20x20), variable: KAMERAREMOTE.bKameraPartDetect, style: Lamp-Lamp1-Green
    Label (40,230 210x20), "Kamera Part Detected"
    Lamp1 (10,250 20x20), variable: KAMERAREMOTE.bKameraAllPass, style: Lamp-Lamp1-Green
    Label (40,250 210x20), "Kamera All pass"
    Lamp1 (10,270 20x20), variable: KAMERAREMOTE.bKameraAnyFail, style: Lamp-Lamp1-Green
    Label (40,270 210x20), "Kamera Any fail"
    Lamp1 (10,300 20x20), variable: KAMERAREMOTE.bKameraOut04, style: Lamp-Lamp1-Green
    Label (40,300 210x20), "Kamera Adapter"
    Lamp1 (10,320 20x20), variable: KAMERAREMOTE.bKameraOut05, style: Lamp-Lamp1-Green
    Label (40,320 210x20), "Kamera Kappe"
    Button (290,290 120x40), "Kamera Run"
        toggle KameraProcess.bKameraRun
    Button (530,290 100x50), "Checker indítása", tooltip "A Pt oldali kamera saját vezérlő szoftvere", pressed state: Laser.bStartFOBADraw
        OnMouseUp: execute { KAMERAREMOTE.bStartChecker:=TRUE; }
END_VISUALIZATION

// ---- VISUs/Login.TcVIS
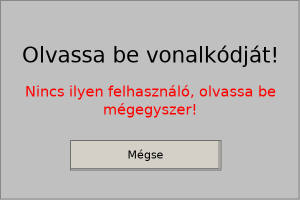
VISUALIZATION Login  // 300x200
    Label (10,40 281x30), "Olvassa be vonalkódját!"
    Button (70,140 151x30), "Mégse"
        toggle GVL.LoginEnabled
    Label (10,80 281x41), "Nincs ilyen felhasználó, olvassa be mégegyszer!", invisible if: NOT GVL.UserNotFound
END_VISUALIZATION

// ---- VISUs/Pt1000_oldali_kamera.TcVIS
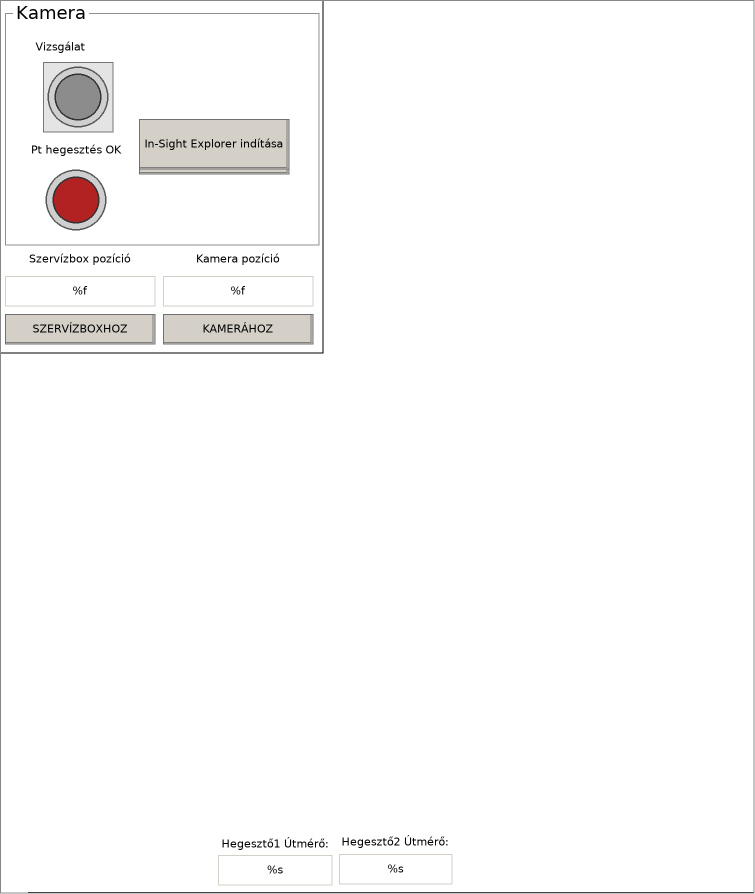
VISUALIZATION Pt1000_oldali_kamera  // 755x894
    Rectangle (0,0 323x353)
    Textfield (218,855 114x30), "%s", text variable: HEGESZTOK.ulHegeszto1Utmero, input disabled if: TRUE
    Label (200,829 150x30), "Hegesztő1 Útmérő:"
    Textfield (339,854 113x30), "%s", text variable: HEGESZTOK.ulHegeszto2Utmero, input disabled if: TRUE
    Label (320,827 150x30), "Hegesztő2 Útmérő:"
    Line (28,892) (753,892)
    GroupBox (5,5 314x240), "Kamera"
        PushSwitch (38,57 70x70), variable: GVL.bPtKameraTrigger, behaviour: TOGGLE, style: Switch-PushSwitch-Gray
        Label (22,32 67x20), "Vizsgálat"
        Button (134,119 150x50), "IV-Navigator indítása", tooltip "A jelölö lézer saját vezérlö szoftvere", pressed state: Laser.bStartFOBADraw
            OnMouseUp: execute { KAMERA.bStartIVNav:=TRUE; }
        Group (18,135 106x95)
            Label (0,0 106x20), "Pt hegesztés OK"
            Lamp1 (18,25 70x70), variable: GVL.bPtKameraHegesztesOK, style: Lamp-Lamp1-Green
            Lamp1 (18,25 70x70), variable: NOT GVL.bPtKameraHegesztesOK, invisible if: GVL.bPtKameraTrigger OR GVL.bPtKameraHegesztesOK, style: Lamp-Lamp1-Red
        Button (134,114 150x50), "In-Sight Explorer indítása", tooltip "A jelölö lézer saját vezérlö szoftvere", pressed state: Laser.bStartFOBADraw
            OnMouseUp: ExecuteCommand ExecuteCommand=ExecuteCommand=[Command=ExecuteClientProgram, Value='C:\Program Files\Cognex\In-Sight\In-Sight Explorer 5.5.0\In-Sight Explorer.exe']
    Textfield (5,276 150x30), "%f", text variable: GVL.lrPtSzervizbox
    Button (5,314 150x30), "SZERVÍZBOXHOZ"
        OnMouseUp: execute { PISTITENGELY.lrPistiPosition:=GVL.lrPtSzervizbox; PISTITENGELY.sPistiAxisCommand:='MOVE'; }
    Label (5,249 150x20), "Szervízbox pozíció"
    Textfield (163,276 150x30), "%f", text variable: GVL.lrPtKameraPosition
        OnMouseClick: write the text variable via VisuDialogs.Numpad, min -10000, max -1
    Button (163,314 150x30), "KAMERÁHOZ"
        OnMouseUp: execute { PISTITENGELY.lrPistiPosition:=GVL.lrPtKameraPosition; PISTITENGELY.sPistiAxisCommand:='MOVE'; }
    Label (163,249 150x20), "Kamera pozíció"
END_VISUALIZATION

// ---- VISUs/Hegeszto_statusz.TcVIS
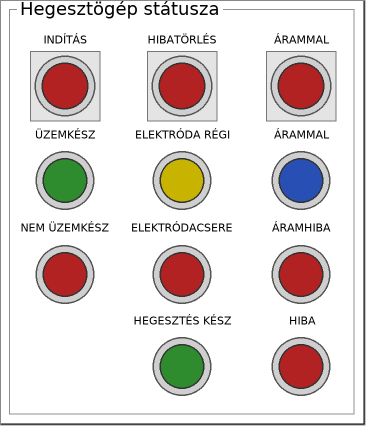
VISUALIZATION Hegeszto_statusz  // 366x426
    Rectangle (0,0 364x424)
    GroupBox (9,1 345x413), "Hegesztögép státusza"
        PushSwitch (138,50 70x70), variable: GVL.bHegesztoHibaTorles, behaviour: TOGGLE, style: Switch-PushSwitch-Red
        PushSwitch (21,50 70x70), variable: HEGESZTOK.bHegesztoStart, behaviour: TOGGLE, style: Switch-PushSwitch-Red
        Label (133,29 80x20), "HIBATÖRLÉS"
        Label (258,29 69x20), "ÁRAMMAL"
        Lamp1 (139,145 68x69), variable: HEGESZTOK.bHegesztoVorwarnung, style: Lamp-Lamp1-Yellow
        Lamp1 (139,239 68x69), variable: HEGESZTOK.bHegesztoElektrodenAnfordem, style: Lamp-Lamp1-Red
        Lamp1 (22,145 68x69), variable: HEGESZTOK.bHegesztoBereit, style: Lamp-Lamp1-Green
        Lamp1 (258,239 68x69), variable: HEGESZTOK.bHegesztoStromFehler, style: Lamp-Lamp1-Red
        Label (258,217 69x20), "ÁRAMHIBA"
        Label (258,124 69x20), "ÁRAMMAL"
        Lamp1 (22,239 68x69), variable: HEGESZTOK.bHegesztoNichtBereit, style: Lamp-Lamp1-Red
        Label (112,124 123x20), "ELEKTRÓDA RÉGI"
        Lamp1 (258,145 68x69), variable: HEGESZTOK.bHegesztoMitStromIn, style: Lamp-Lamp1-Blue
        Label (22,29 69x20), "INDÍTÁS"
        Label (22,124 69x20), "ÜZEMKÉSZ"
        Label (114,217 118x20), "ELEKTRÓDACSERE"
        Label (3,217 106x20), "NEM ÜZEMKÉSZ"
        PushSwitch (257,50 70x70), variable: HEGESZTOK.bHegesztoMitStromOut, behaviour: TOGGLE, style: Switch-PushSwitch-Red
        Lamp1 (258,331 68x69), variable: GVL.bHegesztoHiba, style: Lamp-Lamp1-Red
        Lamp1 (139,331 68x69), variable: HEGESZTOK.bHegesztoFK, style: Lamp-Lamp1-Green
        Label (113,310 121x20), "HEGESZTÉS KÉSZ"
    Label (268,311 69x20), "HIBA"
END_VISUALIZATION

// ---- VISUs/Lezer.TcVIS
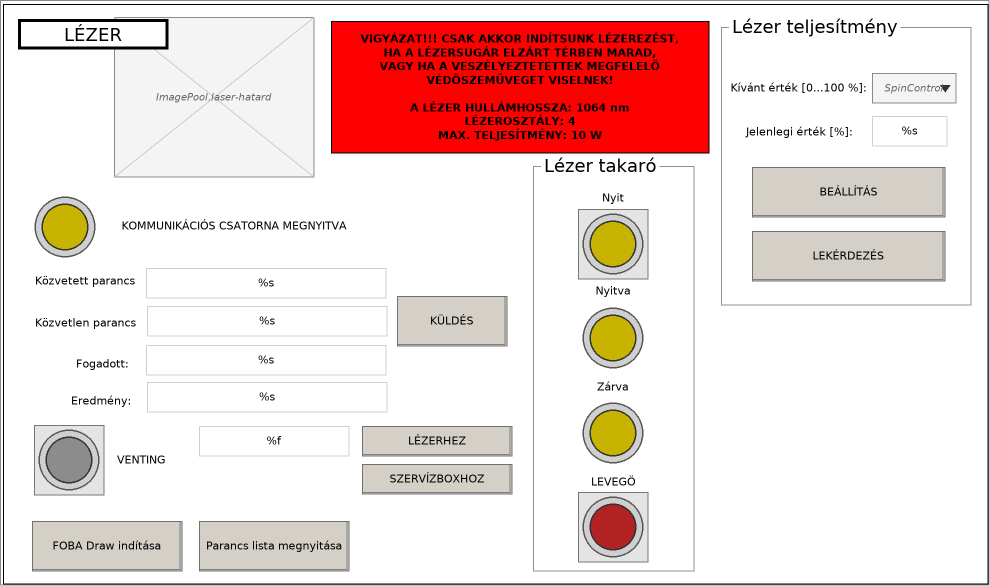
VISUALIZATION Lezer  // 990x586
    Rectangle (3,4 985x580)
    Textfield (146,268 240x30), "%s", text variable: Laser.s_InCommand
        OnMouseClick: write Laser.s_InCommand via VisuDialogs.Keypad
    Textfield (146,345 240x30), "%s", text variable: Laser.sLaserReceived
    Lamp1 (30,192 70x70), variable: GVL.bLaserCommOpen, style: Lamp-Lamp1-Yellow
    Label (106,211 256x30), "KOMMUNIKÁCIÓS CSATORNA MEGNYITVA"
    Label (70,349 65x30), "Fogadott:"
    PushSwitch (34,425 70x70), variable: AUTOMATA.bElszivasBe, behaviour: TOGGLE, style: Switch-PushSwitch-Gray
    Label (110,445 63x30), "VENTING"
    Label (24,266 114x30), "Közvetett parancs"
    Label (25,308 114x30), "Közvetlen parancs"
    Textfield (147,306 240x30), "%s", text variable: Laser.sLaserSend
        OnMouseClick: write Laser.sLaserSend via VisuDialogs.Keypad
    Button (32,521 150x50), "FOBA Draw indítása", tooltip "A jelölö lézer saját vezérlö szoftvere", pressed state: Laser.bStartFOBADraw
        OnMouseUp: execute { Laser.bStartFOBADraw:=TRUE; }
    Button (397,296 110x50), "KÜLDÉS"
        OnMouseUp: execute { Laser.iState:=1; }
    Textfield (199,426 150x30), "%f", text variable: GVL.lrVegmeroPosition
        OnMouseClick: write the text variable via VisuDialogs.Numpad, min -10000, max -1
    Image (114,17 200x160), image: ImagePool.laser-hatard
    RoundedRectangle (18,19 150x30)
    Label (18,20 150x30), "LÉZER"
    Button (199,521 150x50), "Parancs lista megnyitása", tooltip "Ultimate script-ben megírt parancsok pdf-ben", pressed state: Laser.bStartUltimate
        OnMouseUp: execute { Laser.bStartUltimate:=TRUE; }
    GroupBox (533,158 161x413), "Lézer takaró"
        PushSwitch (45,51 70x70), variable: VEGMERO.bLezertakaro, behaviour: TOGGLE, style: Switch-PushSwitch-Yellow
        Label (55,30 50x20), "Nyit"
        Lamp1 (45,145 70x70), variable: VEGMERO.bLezertakaroNyitva, style: Lamp-Lamp1-Yellow
        Label (55,123 50x20), "Nyitva"
        Lamp1 (45,240 70x70), variable: VEGMERO.bLezertakaroZarva, style: Lamp-Lamp1-Yellow
        Label (55,219 50x20), "Zárva"
        Group (45,309 70x95)
            PushSwitch (0,25 70x70), variable: MAIN.bLevego, behaviour: TOGGLE, style: Switch-PushSwitch-Red
            Label (1,0 69x30), "LEVEGÖ"
    RoundedRectangle (331,21 378x132), "VIGYÁZAT!!! CSAK AKKOR INDÍTSUNK LÉZEREZÉST, HA A LÉZERSUGÁR ELZÁRT TÉRBEN MARAD, VAGY HA A VESZÉLYEZTETETTEK MEGFELELÖ VÉDÖSZEMÜVEGET VISELNEK! A LÉZER HULLÁMHOSSZA: 1064 nm LÉZEROSZTÁLY: 4 MAX. TELJESÍTMÉNY: 10 W"
    Button (362,426 150x30), "LÉZERHEZ"
        OnMouseUp: execute { PISTITENGELY.lrPistiPosition:=GVL.lrVegmeroPosition; PISTITENGELY.sPistiAxisCommand:='MOVE'; }
    Button (362,464 150x30), "SZERVÍZBOXHOZ"
        OnMouseUp: execute { PISTITENGELY.lrPistiPosition:=GVL.lrPtSzervizbox; PISTITENGELY.sPistiAxisCommand:='MOVE'; }
    Textfield (147,382 240x30), "%s", text variable: Laser.sLaserReceived
    Label (66,386 70x30), "Eredmény:"
    GroupBox (721,19 250x286), "Lézer teljesítmény"
        SpinControl (151,54 84x30), variable: Laser.iWishPower
            OnMouseClick: write Laser.iWishPower via VisuDialogs.Numpad, min 0, max 100
        Label (11,54 133x30), "Kívánt érték [0...100 %]:"
        Label (12,98 133x30), "Jelenlegi érték [%]:"
        Textfield (151,97 75x30), "%s", text variable: Laser.iSetPower
        Button (31,148 193x50), "BEÁLLÍTÁS"
            OnMouseUp: execute {
                Laser.sLaserSend:=CONCAT('SetIntensity;',
                				  CONCAT(INT_TO_STRING(Laser.iWishPower),';'));
                Laser.iState:=1;
            }
        Button (31,212 193x50), "LEKÉRDEZÉS"
            OnMouseUp: execute { Laser.sLaserSend:='GetIntensity;'; Laser.iState:=1; }
END_VISUALIZATION

// ---- VISUs/Kamera.TcVIS
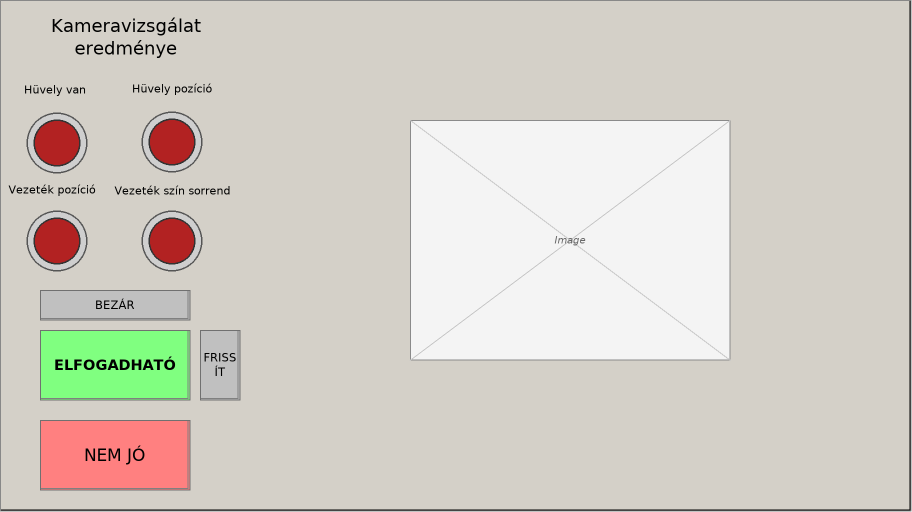
VISUALIZATION Kamera  // 912x512
    Rectangle (0,0 910x510)
    Button (40,420 150x70), "NEM JÓ", invisible if: GVL.bNTCEredmenyGombokRejtve
        OnMouseUp: execute {
            GVL.bNTCKameraNemJo:=TRUE;
            GVL.bNTCEredmenyGombokRejtve:=TRUE;
            GVL.bKameraEredmenyekRejtve:=TRUE;
        }
    Label (10,80 90x20), "Hüvely van"
    Lamp1 (22,108 70x70), variable: GVL.bKameraHulseVanOK, style: Lamp-Lamp1-Green
    Lamp1 (22,108 70x70), variable: NOT GVL.bKameraHulseVanOK, invisible if: NOT KAMERA.bVizsgalatKesz OR GVL.bKameraHulseVanOK, style: Lamp-Lamp1-Red
    Lamp1 (137,107 70x70), variable: GVL.bKameraHulsePozOK, style: Lamp-Lamp1-Green
    Lamp1 (137,206 70x70), variable: GVL.bKameraSzinekOK, style: Lamp-Lamp1-Green
    Label (108,181 129x20), "Vezeték szín sorrend"
    Label (130,80 84x18), "Hüvely pozíció"
    Lamp1 (137,107 70x70), variable: NOT GVL.bKameraHulsePozOK, invisible if: NOT KAMERA.bVizsgalatKesz OR GVL.bKameraHulsePozOK, style: Lamp-Lamp1-Red
    Lamp1 (137,206 70x70), variable: NOT GVL.bKameraSzinekOK, invisible if: NOT KAMERA.bVizsgalatKesz OR GVL.bKameraSzinekOK, style: Lamp-Lamp1-Red
    Label (0,180 104x20), "Vezeték pozíció"
    Lamp1 (22,206 70x70), variable: GVL.bKameraVezetekPozOK, style: Lamp-Lamp1-Green
    Lamp1 (22,206 70x70), variable: NOT GVL.bKameraVezetekPozOK, invisible if: NOT KAMERA.bVizsgalatKesz OR GVL.bKameraVezetekPozOK, style: Lamp-Lamp1-Red
    Label (51,10 150x54), "Kameravizsgálat eredménye"
    Button (40,330 150x70), "ELFOGADHATÓ", invisible if: GVL.bNTCEredmenyGombokRejtve
        OnMouseUp: execute {
            GVL.bNTCKameraElfogadva:=TRUE;
            GVL.bNTCEredmenyGombokRejtve:=TRUE;
            GVL.bKameraEredmenyekRejtve:=TRUE;
        }
    Button (40,290 150x30), "BEZÁR", invisible if: GVL.bNTCBezarGombRejtve
        OnMouseUp: execute {
            //GVL.bNTCBezarGombRejtve:=TRUE;
            GVL.bKameraEredmenyekRejtve:=TRUE;
        }
    Button (200,330 40x70), "FRISSÍT"
        OnMouseUp: execute { GVL.iBitmap_Version:= GVL.iBitmap_Version+1; }
    Image (410,120 320x240)
        p871682116: GVL.iBitmap_Version
        p84334746: GVL.sNTCKameraImageID
END_VISUALIZATION

// ---- VISUs/Robot.TcVIS
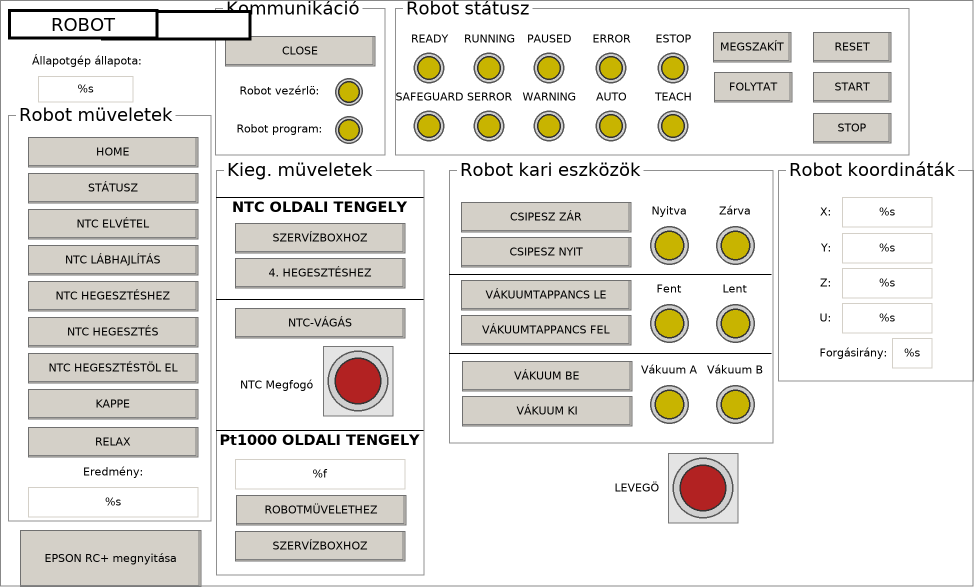
VISUALIZATION Robot  // 974x587
    GroupBox (215,0 170x155), "Kommunikáció"
        Button (10,36 150x30), "OPEN", invisible if: RobotProcess.iState>0, input disabled if: RobotProcess.iState>0
            OnMouseClick: execute { RobotProcess.iState:=1; }
        Button (10,36 150x30), "CLOSE", invisible if: RobotProcess.iState=0, input disabled if: RobotProcess.iState=0
            OnMouseClick: execute { RobotProcess.iState:=200; }
        Lamp1 (116,76 36x32), variable: ROBOTREMOTE.bRobotCommOpen, style: Lamp-Lamp1-Yellow
        Label (23,81 84x20), "Robot vezérlö:"
        Label (9,119 101x20), "Robot program:"
        Lamp1 (116,114 36x32), variable: ROBOTCOMMAND.bRobotCommOpen, style: Lamp-Lamp1-Yellow
    GroupBox (395,0 514x155), "Robot státusz", invisible if: RobotProcess.iState=0, input disabled if: RobotProcess.iState=0
        Lamp1 (16,50 36x36), variable: RobotProcess.baStatus[10], invisible if: ROBOTREMOTE.bRobotCommOpen=FALSE, style: Lamp-Lamp1-Yellow
        Label (6,24 57x30), "READY", invisible if: ROBOTREMOTE.bRobotCommOpen=FALSE
        Lamp1 (76,50 36x36), variable: RobotProcess.baStatus[9], invisible if: ROBOTREMOTE.bRobotCommOpen=FALSE, style: Lamp-Lamp1-Yellow
        Label (66,24 57x30), "RUNNING", invisible if: ROBOTREMOTE.bRobotCommOpen=FALSE
        Lamp1 (136,50 36x36), variable: RobotProcess.baStatus[8], invisible if: ROBOTREMOTE.bRobotCommOpen=FALSE, style: Lamp-Lamp1-Yellow
        Label (126,24 57x30), "PAUSED", invisible if: ROBOTREMOTE.bRobotCommOpen=FALSE
        Lamp1 (198,50 36x36), variable: RobotProcess.baStatus[7], invisible if: ROBOTREMOTE.bRobotCommOpen=FALSE, style: Lamp-Lamp1-Yellow
        Label (188,24 57x30), "ERROR", invisible if: ROBOTREMOTE.bRobotCommOpen=FALSE
        Lamp1 (260,50 36x36), variable: RobotProcess.baStatus[6], invisible if: ROBOTREMOTE.bRobotCommOpen=FALSE, style: Lamp-Lamp1-Yellow
        Label (250,24 57x30), "ESTOP", invisible if: ROBOTREMOTE.bRobotCommOpen=FALSE
        Lamp1 (16,108 36x36), variable: RobotProcess.baStatus[5], invisible if: ROBOTREMOTE.bRobotCommOpen=FALSE, style: Lamp-Lamp1-Yellow
        Label (6,82 57x30), "SAFEGUARD", invisible if: ROBOTREMOTE.bRobotCommOpen=FALSE
        Lamp1 (76,108 36x36), variable: RobotProcess.baStatus[4], invisible if: ROBOTREMOTE.bRobotCommOpen=FALSE, style: Lamp-Lamp1-Yellow
        Label (66,82 57x30), "SERROR", invisible if: ROBOTREMOTE.bRobotCommOpen=FALSE
        Lamp1 (136,108 36x36), variable: RobotProcess.baStatus[3], invisible if: ROBOTREMOTE.bRobotCommOpen=FALSE, style: Lamp-Lamp1-Yellow
        Label (126,82 57x30), "WARNING", invisible if: ROBOTREMOTE.bRobotCommOpen=FALSE
        Lamp1 (198,108 36x36), variable: RobotProcess.baStatus[2], invisible if: ROBOTREMOTE.bRobotCommOpen=FALSE, style: Lamp-Lamp1-Yellow
        Label (188,82 57x30), "AUTO", invisible if: ROBOTREMOTE.bRobotCommOpen=FALSE
        Lamp1 (260,108 36x36), variable: RobotProcess.baStatus[1], invisible if: ROBOTREMOTE.bRobotCommOpen=FALSE, style: Lamp-Lamp1-Yellow
        Label (250,82 57x30), "TEACH", invisible if: ROBOTREMOTE.bRobotCommOpen=FALSE
        RoundedRectangle (-294,10 150x30)
        Button (318,32 78x30), "MEGSZAKÍT"
            OnMouseClick: execute { ROBOTREMOTE.sRobotCommand := 'Pause'; ROBOTREMOTE.bRobotCommandSend := TRUE; }
        Button (319,72 78x30), "FOLYTAT"
            OnMouseClick: execute { ROBOTREMOTE.sRobotCommand := 'Continue'; ROBOTREMOTE.bRobotCommandSend := TRUE; }
        Button (418,32 78x30), "RESET"
            OnMouseClick: execute { ROBOTREMOTE.sRobotCommand := 'Reset'; ROBOTREMOTE.bRobotCommandSend := TRUE; }
        Button (418,72 78x30), "START"
            OnMouseClick: execute {
                ROBOTREMOTE.sRobotCommand := 'Start';
                ROBOTREMOTE.sRobotCommandParam1 := '0';
                ROBOTREMOTE.bRobotCommandSend := TRUE;
            }
        Button (418,113 78x30), "STOP"
            OnMouseClick: execute { ROBOTREMOTE.sRobotCommand := 'Stop'; ROBOTREMOTE.bRobotCommandSend := TRUE; }
    GroupBox (8,107 203x414), "Robot müveletek", invisible if: RobotProcess.iState=0, input disabled if: RobotProcess.iState=0
        Button (20,102 170x30), "NTC ELVÉTEL", invisible if: RobotProcess.iState=0, input disabled if: RobotProcess.iState=0
            OnMouseClick: execute { RobotProcess.s_InRobotTCPCommand := 'NTCHEZ'; }
        Button (20,174 170x30), "NTC HEGESZTÉSHEZ", invisible if: RobotProcess.iState=0, input disabled if: RobotProcess.iState=0
            OnMouseClick: execute { RobotProcess.s_InRobotTCPCommand := 'NTCHEG'; }
        Button (20,246 170x30), "NTC HEGESZTÉSTÖL EL", invisible if: RobotProcess.iState=0, input disabled if: RobotProcess.iState=0
            OnMouseClick: execute { RobotProcess.s_InRobotTCPCommand := 'NTCHEGTOL'; }
        Button (20,282 170x30), "KAPPE", invisible if: RobotProcess.iState=0, input disabled if: RobotProcess.iState=0
            OnMouseClick: execute { RobotProcess.s_InRobotTCPCommand := 'KAPPE'; }
        Button (20,320 170x30), "RELAX", invisible if: RobotProcess.iState=0, input disabled if: RobotProcess.iState=0
            OnMouseClick: execute { RobotProcess.s_InRobotTCPCommand := 'RELAX'; }
        Button (20,30 170x30), "HOME", invisible if: RobotProcess.iState=0, input disabled if: RobotProcess.iState=0
            OnMouseClick: execute { RobotProcess.s_InRobotTCPCommand := 'HOME'; }
        Textfield (20,380 170x30), "%s", text variable: ROBOTCOMMAND.sRobotResult, input disabled if: TRUE
        Label (60,350 90x30), "Eredmény:"
        Button (20,138 170x30), "NTC LÁBHAJLÍTÁS", invisible if: RobotProcess.iState=0, input disabled if: RobotProcess.iState=0
            OnMouseClick: execute { RobotProcess.s_InRobotTCPCommand := 'NTCLAB'; }
        Button (20,66 170x30), "STÁTUSZ", invisible if: RobotProcess.iState=0, input disabled if: RobotProcess.iState=0
            OnMouseClick: execute { RobotProcess.s_InRobotTCPCommand := 'STATUSZ'; }
        Button (20,210 170x30), "NTC HEGESZTÉS", invisible if: RobotProcess.iState=0, input disabled if: RobotProcess.iState=0
            OnMouseClick: execute {
                IF ROBOTCOMMAND.sRobotResult='NTCHEG' THEN
                	RobotProcess.s_InRobotTCPCommand := 'NTCHEG2';
                END_IF
            }
    Textfield (38,76 95x26), "%s", text variable: RobotProcess.iState, input disabled if: TRUE
    GroupBox (216,162 208x413), "Kieg. müveletek", invisible if: RobotProcess.iState=0, input disabled if: RobotProcess.iState=0
        Button (19,146 170x30), "NTC-VÁGÁS", input disabled if: NTCProcess.s_InCommand <> ''
            OnMouseUp: execute {
                IF NTCProcess.s_InCommand = '' THEN
                	NTCProcess.s_InCommand:='VAGAS';
                END_IF
            }
        Button (19,96 170x30), "4. HEGESZTÉSHEZ"
            OnMouseUp: execute { JOZSITENGELY.lrJozsiPosition:=GVL.lrHegesztoPosition4; JOZSITENGELY.sJozsiAxisCommand:='MOVE'; }
        PushSwitch (107,184 70x70), variable: NTCProcess.bMegfogo, behaviour: TOGGLE, style: Switch-PushSwitch-Red
        Label (17,213 87x20), "NTC Megfogó"
        Textfield (19,297 170x30), "%f", text variable: GVL.lrRobotKappePosition
            OnMouseClick: write the text variable via VisuDialogs.Numpad, min -10000, max -1
        Button (19,61 170x30), "SZERVÍZBOXHOZ"
            OnMouseUp: execute { JOZSITENGELY.lrJozsiPosition:=GVL.lrNTCSzervizbox; JOZSITENGELY.sJozsiAxisCommand:='MOVE'; }
        Button (19,369 170x30), "SZERVÍZBOXHOZ"
            OnMouseUp: execute { PISTITENGELY.lrPistiPosition:=GVL.lrPtSzervizbox; PISTITENGELY.sPistiAxisCommand:='MOVE'; }
        Line (0,268) (207,268), "Pt1000 OLDALI TENGELY"
        Line (0,35) (207,35), "NTC OLDALI TENGELY"
        Line (0,137) (207,137)
        Button (20,333 170x30), "ROBOTMÜVELETHEZ"
            OnMouseUp: execute { PISTITENGELY.lrPistiPosition:=GVL.lrRobotKappePosition; PISTITENGELY.sPistiAxisCommand:='MOVE'; }
    Label (27,46 120x30), "Állapotgép állapota:"
    RoundedRectangle (8,9 150x30)
    Label (8,10 150x30), "ROBOT"
    GroupBox (449,162 324x281), "Robot kari eszközök", invisible if: RobotProcess.iState=0, input disabled if: RobotProcess.iState=0
        Button (12,40 170x30), "CSIPESZ ZÁR", invisible if: RobotProcess.iState=0, input disabled if: RobotProcess.iState=0
            OnMouseClick: execute { RobotProcess.s_InRobotTCPCommand := 'CSIPESZ_ZAR'; }
        Button (12,75 170x30), "CSIPESZ NYIT", invisible if: RobotProcess.iState=0, input disabled if: RobotProcess.iState=0
            OnMouseClick: execute { RobotProcess.s_InRobotTCPCommand := 'CSIPESZ_NYIT'; }
        Group (12,118 170x65)
            Button (0,0 170x30), "VÁKUUMTAPPANCS LE", invisible if: RobotProcess.iState=0, input disabled if: RobotProcess.iState=0
                OnMouseClick: execute { RobotProcess.s_InRobotTCPCommand := 'SZIPPANTO_LE'; }
            Button (0,35 170x30), "VÁKUUMTAPPANCS FEL", invisible if: RobotProcess.iState=0, input disabled if: RobotProcess.iState=0
                OnMouseClick: execute { RobotProcess.s_InRobotTCPCommand := 'SZIPPANTO_FEL'; }
        Group (13,199 170x65)
            Button (0,35 170x30), "VÁKUUM KI", invisible if: RobotProcess.iState=0, input disabled if: RobotProcess.iState=0
                OnMouseClick: execute { RobotProcess.s_InRobotTCPCommand := 'VAKUUM_KI'; }
            Button (0,0 170x30), "VÁKUUM BE", invisible if: RobotProcess.iState=0, input disabled if: RobotProcess.iState=0
                OnMouseClick: execute { RobotProcess.s_InRobotTCPCommand := 'VAKUUM_BE'; }
        Lamp1 (198,61 45x45), variable: GVL.stRobotStatusz.bCsipeszNyitva, style: Lamp-Lamp1-Yellow
        Label (190,39 60x20), "Nyitva"
        Lamp1 (264,61 45x45), variable: GVL.stRobotStatusz.bCsipeszZarva, style: Lamp-Lamp1-Yellow
        Label (256,39 60x20), "Zárva"
        Lamp1 (198,139 45x45), variable: GVL.stRobotStatusz.bVakuumSzippantoFent, style: Lamp-Lamp1-Yellow
        Label (190,117 60x20), "Fent"
        Lamp1 (264,139 45x45), variable: GVL.stRobotStatusz.bVakuumSzippantoLent, style: Lamp-Lamp1-Yellow
        Label (256,117 60x20), "Lent"
        Lamp1 (198,220 45x45), variable: GVL.stRobotStatusz.bVakuumA, style: Lamp-Lamp1-Yellow
        Label (190,198 60x20), "Vákuum A"
        Lamp1 (264,220 45x45), variable: GVL.stRobotStatusz.bVakuumB, style: Lamp-Lamp1-Yellow
        Label (256,198 60x20), "Vákuum B"
        Line (0,112) (322,112)
        Line (0,191) (322,191)
    GroupBox (778,162 196x219), "Robot koordináták", invisible if: RobotProcess.iState=0, input disabled if: RobotProcess.iState=0
        Group (36,35 118x171)
            Label (0,5 20x20), "X:"
            Textfield (28,0 90x30), "%s", text variable: GVL.stRobotStatusz.rX
            Label (0,41 20x20), "Y:"
            Textfield (28,36 90x30), "%s", text variable: GVL.stRobotStatusz.rY
            Label (0,76 20x20), "Z:"
            Textfield (28,71 90x30), "%s", text variable: GVL.stRobotStatusz.rZ
            Textfield (28,106 90x30), "%s", text variable: GVL.stRobotStatusz.rU
            Label (0,111 20x20), "U:"
            Textfield (78,141 40x30), "%s", text variable: GVL.stRobotStatusz.sHand
            Label (0,146 76x20), "Forgásirány:"
    Group (607,453 131x70), invisible if: RobotProcess.iState=0, input disabled if: RobotProcess.iState=0
        PushSwitch (61,0 70x70), variable: MAIN.bLevego, behaviour: TOGGLE, style: Switch-PushSwitch-Red
        Label (0,20 55x30), "LEVEGÖ"
    Button (20,530 181x57), "EPSON RC+ megnyitása"
        OnMouseUp: ExecuteCommand ExecuteCommand=ExecuteCommand=[Command=ExecuteClientProgram, Value='C:\EpsonRC70\exe\erc70.exe']
END_VISUALIZATION

// ---- VISUs/Kappe_pres.TcVIS
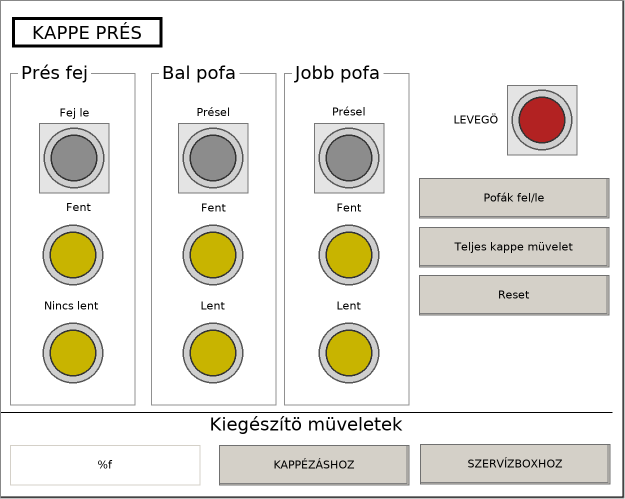
VISUALIZATION Kappe_pres  // 625x499
    Rectangle (0,0 623x497)
    GroupBox (151,65 125x340), "Bal pofa"
        Lamp1 (27,155 70x70), variable: KAPPE.bKappeBalFent, style: Lamp-Lamp1-Yellow
        Label (45,128 35x30), "Fent"
        Lamp1 (27,253 70x70), variable: KAPPE.bKappeBalLent, style: Lamp-Lamp1-Yellow
        Label (43,226 38x30), "Lent"
        PushSwitch (27,58 70x70), variable: KAPPE.bKappeBalFelLe, behaviour: TOGGLE, style: Switch-PushSwitch-Gray
        Label (37,33 51x29), "Présel"
    Button (419,178 190x40), "Pofák fel/le", input disabled if: KAPPE.bKappeBalFent<>KAPPE.bKappeJobbFent AND KAPPE.bKappeBalLent<>KAPPE.bKappeJobbLent
        OnMouseUp: execute {
            IF ((KAPPE.bKappeBalFent=TRUE) AND (KAPPE.bKappeBalLent=FALSE) AND (KAPPE.bKappeJobbFent=TRUE) AND (KAPPE.bKappeJobbLent=FALSE)) THEN
            	KAPPE.bKappeBalFelLe:=TRUE;
            	KAPPE.bKappeJobbFelLe:=TRUE;
            ELSE
            	KAPPE.bKappeBalFelLe:=FALSE;
            	KAPPE.bKappeJobbFelLe:=FALSE;
            END_IF
        }
    Button (419,227 190x40), "Teljes kappe müvelet", input disabled if: KAPPE.bKappeBalFent<>KAPPE.bKappeJobbFent AND KAPPE.bKappeBalLent<>KAPPE.bKappeJobbLent
        OnMouseUp: execute { KAPPE.s_InCommand:='START'; }
    GroupBox (284,65 125x340), "Jobb pofa"
        Lamp1 (30,155 70x70), variable: KAPPE.bKappeJobbFent, style: Lamp-Lamp1-Yellow
        Label (47,128 36x30), "Fent"
        Lamp1 (30,253 70x70), variable: KAPPE.bKappeJobbLent, style: Lamp-Lamp1-Yellow
        Label (46,226 38x30), "Lent"
        PushSwitch (30,58 70x70), variable: KAPPE.bKappeJobbFelLe, behaviour: TOGGLE, style: Switch-PushSwitch-Gray
        Label (41,32 48x30), "Présel"
    GroupBox (10,65 125x340), "Prés fej"
        Lamp1 (28,253 70x70), variable: GVL.bKappepresNincsLegalul, style: Lamp-Lamp1-Yellow
        Label (28,226 67x30), "Nincs lent"
        PushSwitch (29,58 70x70), variable: KAPPE.bKappeFelLe, behaviour: TOGGLE, style: Switch-PushSwitch-Gray
        Label (28,33 73x30), "Fej le"
        Lamp1 (28,155 70x70), variable: GVL.bKappePresFent, style: Lamp-Lamp1-Yellow
        Label (32,128 73x29), "Fent"
    RoundedRectangle (12,17 150x30)
    Label (12,18 150x30), "KAPPE PRÉS"
    Textfield (10,445 190x40), "%f", text variable: GVL.lrKappePosition
        OnMouseClick: write the text variable via VisuDialogs.Numpad, min -10000, max -1
    Button (219,445 190x40), "KAPPÉZÁSHOZ"
        OnMouseUp: execute { PISTITENGELY.lrPistiPosition:=GVL.lrKappePosition; PISTITENGELY.sPistiAxisCommand:='MOVE'; }
    Button (420,444 190x40), "SZERVÍZBOXHOZ"
        OnMouseUp: execute { PISTITENGELY.lrPistiPosition:=GVL.lrPtSzervizbox; PISTITENGELY.sPistiAxisCommand:='MOVE'; }
    Line (0,412) (612,412), "Kiegészítö müveletek"
    Group (446,85 131x70)
        PushSwitch (61,0 70x70), variable: MAIN.bLevego, behaviour: TOGGLE, style: Switch-PushSwitch-Red
        Label (0,20 55x30), "LEVEGÖ"
    Button (419,275 190x40), "Reset"
        OnMouseUp: execute { KAPPE.s_InCommand:='RESET'; }
END_VISUALIZATION

// ---- VISUs/Start_ablak.TcVIS
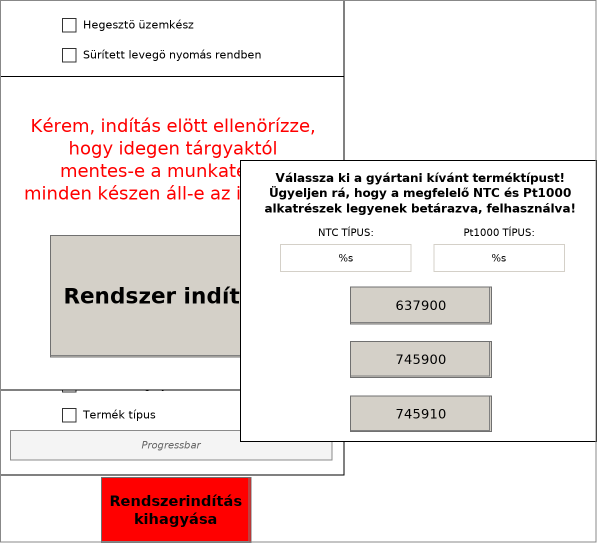
VISUALIZATION Start_ablak  // 597x543
    RoundedRectangle (0,0 344x475)
    Frame (60,10 239x320)
        shows Start_ellenorzes()
    Group (0,76 344x314), invisible if: INIT.iState>0
        RoundedRectangle (0,0 344x314), invisible if: INIT.iState>0, input disabled if: INIT.iState>0
        Label (13,21 320x125), "Kérem, indítás elött ellenörízze, hogy idegen tárgyaktól mentes-e a munkatér, és minden készen áll-e az indításra!"
        Button (50,159 246x122), "Rendszer indítása", invisible if: INIT.iState>0, input disabled if: INIT.iState>0
            OnMouseClick: execute { INIT.iState:=1; }
    Button (101,477 150x66), "Rendszerindítás kihagyása"
        OnMouseClick: execute {
            INIT.iState:=5;
            GVL.bSystemStarted:=TRUE;
            GVL.bSystemNotStarted:=FALSE;
        }
    Progressbar (10,430 322x30), variable: INIT.iKeszenletFoka, invisible if: GVL.bSystemStarted
    Frame (240,160 357x291)
        shows Termektipus()
END_VISUALIZATION

